LIN {X 0,Y 149.107,Z 804.963,A -85,B 0,C 180,E1 -24968.646,E2 -24968.646} C_VEL
LIN {X 0,Y 155.248,Z 796.631,A -85,B 0,C 180,E1 -24971.89,E2 -24971.89} C_VEL
LIN {X 0,Y 160.793,Z 788.072,A -85,B 0,C 180,E1 -24974.372,E2 -24974.372} C_VEL
LIN {X 0,Y 166.724,Z 777.561,A -85,B 0,C 180,E1 -24976.646,E2 -24976.646} C_VEL
LIN {X 0,Y 171.709,Z 767.159,A -85,B 0,C 180,E1 -24978.327,E2 -24978.327} C_VEL
LIN {X 0,Y 176.218,Z 755.637,A -85,B 0,C 180,E1 -24979.706,E2 -24979.706} C_VEL
LIN {X 0,Y 180.103,Z 742.538,A -85,B 0,C 180,E1 -24980.855,E2 -24980.855} C_VEL
LIN {X 0,Y 182.778,Z 729.709,A -85,B 0,C 180,E1 -24981.625,E2 -24981.625} C_VEL
LIN {X 0,Y 184.427,Z 715.563,A -85,B 0,C 180,E1 -24982.173,E2 -24982.173} C_VEL
LIN {X 0,Y 185.741,Z 699.59,A -85,B 0,C 180,E1 -24982.676,E2 -24982.676} C_VEL
LIN {X 0,Y 185.63,Z 687.899,A -85,B 0,C 180,E1 -24983.577,E2 -24983.577} C_VEL
LIN {X 0,Y 184.651,Z 684.228,A -85,B 0,C 180,E1 -24984.352,E2 -24984.352} C_VEL
LIN {X 0,Y 180.191,Z 675.322,A -85,B 0,C 180,E1 -24987.593,E2 -24987.593} C_VEL
LIN {X 0,Y 176.995,Z 669.722,A -85,B 0,C 180,E1 -24990.207,E2 -24990.207} C_VEL
LIN {X 0,Y 173.204,Z 663.907,A -85,B 0,C 180,E1 -24993.751,E2 -24993.751} C_VEL
LIN {X 0,Y 170.669,Z 660.092,A -85,B 0,C 180,E1 -24996.576,E2 -24996.576} C_VEL
LIN {X 0,Y 168.154,Z 656.304,A -85,B 0,C 180,E1 -24999.989,E2 -24999.989} C_VEL
LIN {X 0,Y 165.387,Z 652.572,A -85,B 0,C 180,E1 -25005.228,E2 -25005.228} C_VEL
LIN {X 0,Y 164.803,Z 650.964,A -85,B 0,C 180,E1 -25007.063,E2 -25007.063} C_VEL
LIN {X 0,Y 163.574,Z 650.195,A -85,B 0,C 180,E1 -25012.594,E2 -25012.594} C_VEL
LIN {X 0,Y 163.96,Z 650.175,A -85,B 0,C 180,E1 -25018.772,E2 -25018.772} C_VEL
LIN {X 0,Y 165.067,Z 651.088,A -85,B 0,C 180,E1 -25022.589,E2 -25022.589} C_VEL
LIN {X 0,Y 166.617,Z 654.282,A -85,B 0,C 180,E1 -25026.357,E2 -25026.357} C_VEL
LIN {X 0,Y 168.172,Z 656.106,A -85,B 0,C 180,E1 -25028.941,E2 -25028.941} C_VEL
LIN {X 0,Y 170.766,Z 660.079,A -85,B 0,C 180,E1 -25032.478,E2 -25032.478} C_VEL
LIN {X 0,Y 174.551,Z 665.825,A -85,B 0,C 180,E1 -25036.521,E2 -25036.521} C_VEL
LIN {X 0,Y 178.449,Z 672.031,A -85,B 0,C 180,E1 -25039.947,E2 -25039.947} C_VEL
LIN {X 0,Y 183.117,Z 680.317,A -85,B 0,C 180,E1 -25043.47,E2 -25043.47} C_VEL
LIN {X 0,Y 186.858,Z 687.514,A -85,B 0,C 180,E1 -25045.951,E2 -25045.951} C_VEL
LIN {X 0,Y 185.177,Z 708.656,A -85,B 0,C 180,E1 -25046.819,E2 -25046.819} C_VEL
LIN {X 0,Y 183.07,Z 721.345,A -85,B 0,C 180,E1 -25047.63,E2 -25047.63} C_VEL
LIN {X 0,Y 179.924,Z 734.079,A -85,B 0,C 180,E1 -25048.788,E2 -25048.788} C_VEL
LIN {X 0,Y 176.07,Z 745.896,A -85,B 0,C 180,E1 -25050.327,E2 -25050.327} C_VEL
LIN {X 0,Y 171.395,Z 757.092,A -85,B 0,C 180,E1 -25052.213,E2 -25052.213} C_VEL
LIN {X 0,Y 166.178,Z 767.268,A -85,B 0,C 180,E1 -25054.444,E2 -25054.444} C_VEL
LIN {X 0,Y 160.701,Z 776.286,A -85,B 0,C 180,E1 -25057.05,E2 -25057.05} C_VEL
LIN {X 0,Y 155.565,Z 783.661,A -85,B 0,C 180,E1 -25059.826,E2 -25059.826} C_VEL
LIN {X 0,Y 149.854,Z 790.842,A -85,B 0,C 180,E1 -25063.372,E2 -25063.372} C_VEL
LIN {X 0,Y 144.674,Z 796.477,A -85,B 0,C 180,E1 -25067.15,E2 -25067.15} C_VEL
LIN {X 0,Y 140.117,Z 800.824,A -85,B 0,C 180,E1 -25071.174,E2 -25071.174} C_VEL
LIN {X 0,Y 135.784,Z 804.333,A -85,B 0,C 180,E1 -25075.908,E2 -25075.908} C_VEL
LIN {X 0,Y 132.074,Z 806.745,A -85,B 0,C 180,E1 -25081.386,E2 -25081.386} C_VEL
LIN {X 0,Y 129.344,Z 807.693,A -85,B 0,C 180,E1 -25087.475,E2 -25087.475} C_VEL
LIN {X 0,Y 128.338,Z 807.582,A -85,B 0,C 180,E1 -25090.819,E2 -25090.819} C_VEL
LIN {X 0,Y 127.671,Z 807.045,A -85,B 0,C 180,E1 -25094.024,E2 -25094.024} C_VEL
LIN {X 0,Y 127.38,Z 806.076,A -85,B 0,C 180,E1 -25097.251,E2 -25097.251} C_VEL
LIN {X 0,Y 127.514,Z 803.466,A -85,B 0,C 180,E1 -25102.784,E2 -25102.784} C_VEL
LIN {X 0,Y 128.551,Z 799.409,A -85,B 0,C 180,E1 -25108.434,E2 -25108.434} C_VEL
LIN {X 0,Y 129.967,Z 794.796,A -85,B 0,C 180,E1 -25113.1,E2 -25113.1} C_VEL
LIN {X 0,Y 132.074,Z 788.942,A -85,B 0,C 180,E1 -25117.645,E2 -25117.645} C_VEL
LIN {X 0,Y 134.811,Z 781.651,A -85,B 0,C 180,E1 -25122.036,E2 -25122.036} C_VEL
LIN {X 0,Y 137.595,Z 774.209,A -85,B 0,C 180,E1 -25125.554,E2 -25125.554} C_VEL
LIN {X 0,Y 139.505,Z 769.017,A -85,B 0,C 180,E1 -25127.593,E2 -25127.593} C_VEL
LIN {X 0,Y 137.283,Z 767.608,A -85,B 0,C 180,E1 -25128.723,E2 -25128.723} C_VEL
LIN {X 0,Y 136.619,Z 766.743,A -85,B 0,C 180,E1 -25129.295,E2 -25129.295} C_VEL
LIN {X 0,Y 133.731,Z 776.449,A -85,B 0,C 180,E1 -25133.212,E2 -25133.212} C_VEL
LIN {X 0,Y 131.498,Z 784.057,A -85,B 0,C 180,E1 -25137.111,E2 -25137.111} C_VEL
LIN {X 0,Y 129.644,Z 790.883,A -85,B 0,C 180,E1 -25141.489,E2 -25141.489} C_VEL
LIN {X 0,Y 128.29,Z 796.393,A -85,B 0,C 180,E1 -25145.922,E2 -25145.922} C_VEL
LIN {X 0,Y 127.318,Z 801.706,A -85,B 0,C 180,E1 -25151.482,E2 -25151.482} C_VEL
LIN {X 0,Y 127.189,Z 804.837,A -85,B 0,C 180,E1 -25155.915,E2 -25155.915} C_VEL
LIN {X 0,Y 127.664,Z 807.177,A -85,B 0,C 180,E1 -25160.416,E2 -25160.416} C_VEL
LIN {X 0,Y 128.778,Z 808.735,A -85,B 0,C 180,E1 -25164.945,E2 -25164.945} C_VEL
LIN {X 0,Y 130.611,Z 809.478,A -85,B 0,C 180,E1 -25169.419,E2 -25169.419} C_VEL
LIN {X 0,Y 134.05,Z 809.144,A -85,B 0,C 180,E1 -25175.202,E2 -25175.202} C_VEL
LIN {X 0,Y 137.079,Z 808.116,A -85,B 0,C 180,E1 -25178.968,E2 -25178.968} C_VEL
LIN {X 0,Y 142.535,Z 805.212,A -85,B 0,C 180,E1 -25184.265,E2 -25184.265} C_VEL
LIN {X 0,Y 149.024,Z 800.693,A -85,B 0,C 180,E1 -25189.127,E2 -25189.127} C_VEL
LIN {X 0,Y 155.716,Z 794.938,A -85,B 0,C 180,E1 -25193.172,E2 -25193.172} C_VEL
LIN {X 0,Y 161.965,Z 788.671,A -85,B 0,C 180,E1 -25196.368,E2 -25196.368} C_VEL
LIN {X 0,Y 168.681,Z 780.891,A -85,B 0,C 180,E1 -25199.283,E2 -25199.283} C_VEL
LIN {X 0,Y 174.996,Z 772.214,A -85,B 0,C 180,E1 -25201.727,E2 -25201.727} C_VEL
LIN {X 0,Y 181.207,Z 762.147,A -85,B 0,C 180,E1 -25203.892,E2 -25203.892} C_VEL
LIN {X 0,Y 186.728,Z 751.431,A -85,B 0,C 180,E1 -25205.67,E2 -25205.67} C_VEL
LIN {X 0,Y 191.579,Z 739.672,A -85,B 0,C 180,E1 -25207.133,E2 -25207.133} C_VEL
LIN {X 0,Y 195.37,Z 727.803,A -85,B 0,C 180,E1 -25208.273,E2 -25208.273} C_VEL
LIN {X 0,Y 198.233,Z 715.512,A -85,B 0,C 180,E1 -25209.15,E2 -25209.15} C_VEL
LIN {X 0,Y 200.271,Z 701.906,A -85,B 0,C 180,E1 -25209.794,E2 -25209.794} C_VEL
LIN {X 0,Y 201.094,Z 695.258,A -85,B 0,C 180,E1 -25210.064,E2 -25210.064} C_VEL
LIN {X 0,Y 199.845,Z 692.673,A -85,B 0,C 180,E1 -25211.821,E2 -25211.821} C_VEL
LIN {X 0,Y 198.373,Z 689.434,A -85,B 0,C 180,E1 -25214.359,E2 -25214.359} C_VEL
LIN {X 0,Y 197.219,Z 686.711,A -85,B 0,C 180,E1 -25217.375,E2 -25217.375} C_VEL
LIN {X 0,Y 196.404,Z 686.119,A -85,B 0,C 180,E1 -25220.967,E2 -25220.967} C_VEL
LIN {X 0,Y 196.29,Z 687.002,A -85,B 0,C 180,E1 -25223.762,E2 -25223.762} C_VEL
LIN {X 0,Y 196.81,Z 690.184,A -85,B 0,C 180,E1 -25227.513,E2 -25227.513} C_VEL
LIN {X 0,Y 197.265,Z 692.099,A -85,B 0,C 180,E1 -25229.076,E2 -25229.076} C_VEL
LIN {X 0,Y 198.259,Z 696.239,A -85,B 0,C 180,E1 -25231.548,E2 -25231.548} C_VEL
LIN {X 0,Y 199.313,Z 700.889,A -85,B 0,C 180,E1 -25233.671,E2 -25233.671} C_VEL
LIN {X 0,Y 200.13,Z 704.559,A -85,B 0,C 180,E1 -25235.026,E2 -25235.026} C_VEL
LIN {X 0,Y 199.762,Z 708.061,A -85,B 0,C 180,E1 -25235.223,E2 -25235.223} C_VEL
LIN {X 0,Y 197.093,Z 725.443,A -85,B 0,C 180,E1 -25235.867,E2 -25235.867} C_VEL
LIN {X 0,Y 193.859,Z 738.295,A -85,B 0,C 180,E1 -25236.541,E2 -25236.541} C_VEL
LIN {X 0,Y 189.397,Z 751.371,A -85,B 0,C 180,E1 -25237.52,E2 -25237.52} C_VEL
LIN {X 0,Y 184.463,Z 762.701,A -85,B 0,C 180,E1 -25238.646,E2 -25238.646} C_VEL
LIN {X 0,Y 178.307,Z 774.287,A -85,B 0,C 180,E1 -25240.213,E2 -25240.213} C_VEL
LIN {X 0,Y 172.401,Z 783.818,A -85,B 0,C 180,E1 -25241.931,E2 -25241.931} C_VEL
LIN {X 0,Y 164.854,Z 794.256,A -85,B 0,C 180,E1 -25244.434,E2 -25244.434} C_VEL
LIN {X 0,Y 157.908,Z 802.647,A -85,B 0,C 180,E1 -25247.257,E2 -25247.257} C_VEL
LIN {X 0,Y 150.413,Z 810.603,A -85,B 0,C 180,E1 -25250.893,E2 -25250.893} C_VEL
LIN {X 0,Y 144.716,Z 816.086,A -85,B 0,C 180,E1 -25254.355,E2 -25254.355} C_VEL
LIN {X 0,Y 140.343,Z 819.929,A -85,B 0,C 180,E1 -25257.577,E2 -25257.577} C_VEL
LIN {X 0,Y 137.381,Z 821.943,A -85,B 0,C 180,E1 -25259.529,E2 -25259.529} C_VEL
LIN {X 0,Y 131.252,Z 824.616,A -85,B 0,C 180,E1 -25262.665,E2 -25262.665} C_VEL
LIN {X 0,Y 125.55,Z 826.525,A -85,B 0,C 180,E1 -25266.18,E2 -25266.18} C_VEL
LIN {X 0,Y 123.348,Z 827.286,A -85,B 0,C 180,E1 -25268.67,E2 -25268.67} C_VEL
LIN {X 0,Y 121.392,Z 828.217,A -85,B 0,C 180,E1 -25273.174,E2 -25273.174} C_VEL
LIN {X 0,Y 120.096,Z 828.286,A -85,B 0,C 180,E1 -25279.889,E2 -25279.889} C_VEL
LIN {X 0,Y 120.164,Z 827.608,A -85,B 0,C 180,E1 -25283.866,E2 -25283.866} C_VEL
LIN {X 0,Y 120.672,Z 826.255,A -85,B 0,C 180,E1 -25288.749,E2 -25288.749} C_VEL
LIN {X 0,Y 120.78,Z 826.749,A -85,B 0,C 180,E1 -25290,E2 -25290} C_VEL
LIN {X 0,Y 119.997,Z 828.128,A -85,B 0,C 180,E1 -25296.727,E2 -25296.727} C_VEL
LIN {X 0,Y 120.025,Z 828.23,A -85,B 0,C 180,E1 -25300.117,E2 -25300.117} C_VEL
LIN {X 0,Y 121.377,Z 827.211,A -85,B 0,C 180,E1 -25306.828,E2 -25306.828} C_VEL
LIN {X 0,Y 124.481,Z 824.663,A -85,B 0,C 180,E1 -25313.278,E2 -25313.278} C_VEL
LIN {X 0,Y 127.795,Z 821.642,A -85,B 0,C 180,E1 -25317.868,E2 -25317.868} C_VEL
LIN {X 0,Y 131.898,Z 817.615,A -85,B 0,C 180,E1 -25322.196,E2 -25322.196} C_VEL
LIN {X 0,Y 137.817,Z 811.485,A -85,B 0,C 180,E1 -25326.811,E2 -25326.811} C_VEL
LIN {X 0,Y 143.637,Z 804.821,A -85,B 0,C 180,E1 -25330.413,E2 -25330.413} C_VEL
LIN {X 0,Y 150.046,Z 796.598,A -85,B 0,C 180,E1 -25333.698,E2 -25333.698} C_VEL
LIN {X 0,Y 155.805,Z 788.196,A -85,B 0,C 180,E1 -25336.195,E2 -25336.195} C_VEL
LIN {X 0,Y 161.952,Z 777.839,A -85,B 0,C 180,E1 -25338.465,E2 -25338.465} C_VEL
LIN {X 0,Y 167.736,Z 766.224,A -85,B 0,C 180,E1 -25340.343,E2 -25340.343} C_VEL
LIN {X 0,Y 172.414,Z 754.582,A -85,B 0,C 180,E1 -25341.689,E2 -25341.689} C_VEL
LIN {X 0,Y 176.413,Z 741.361,A -85,B 0,C 180,E1 -25342.82,E2 -25342.82} C_VEL
LIN {X 0,Y 179.066,Z 728.861,A -85,B 0,C 180,E1 -25343.542,E2 -25343.542} C_VEL
LIN {X 0,Y 180.73,Z 714.959,A -85,B 0,C 180,E1 -25344.077,E2 -25344.077} C_VEL
LIN {X 0,Y 181.987,Z 699.437,A -85,B 0,C 180,E1 -25344.6,E2 -25344.6} C_VEL
LIN {X 0,Y 181.961,Z 690.827,A -85,B 0,C 180,E1 -25345.285,E2 -25345.285} C_VEL
LIN {X 0,Y 181.33,Z 688.674,A -85,B 0,C 180,E1 -25345.806,E2 -25345.806} C_VEL
LIN {X 0,Y 176.769,Z 679.156,A -85,B 0,C 180,E1 -25349.468,E2 -25349.468} C_VEL
LIN {X 0,Y 173.564,Z 673.777,A -85,B 0,C 180,E1 -25352.365,E2 -25352.365} C_VEL
LIN {X 0,Y 171.058,Z 669.808,A -85,B 0,C 180,E1 -25354.964,E2 -25354.964} C_VEL
LIN {X 0,Y 169.045,Z 666.616,A -85,B 0,C 180,E1 -25357.383,E2 -25357.383} C_VEL
LIN {X 0,Y 166.494,Z 662.608,A -85,B 0,C 180,E1 -25361.159,E2 -25361.159} C_VEL
LIN {X 0,Y 164.281,Z 659.446,A -85,B 0,C 180,E1 -25365.754,E2 -25365.754} C_VEL
LIN {X 0,Y 163.731,Z 657.95,A -85,B 0,C 180,E1 -25367.607,E2 -25367.607} C_VEL
LIN {X 0,Y 162.621,Z 657.234,A -85,B 0,C 180,E1 -25373.703,E2 -25373.703} C_VEL
LIN {X 0,Y 163.082,Z 657.223,A -85,B 0,C 180,E1 -25378.765,E2 -25378.765} C_VEL
LIN {X 0,Y 164.014,Z 658.078,A -85,B 0,C 180,E1 -25382.149,E2 -25382.149} C_VEL
LIN {X 0,Y 165.723,Z 661.5,A -85,B 0,C 180,E1 -25386.391,E2 -25386.391} C_VEL
LIN {X 0,Y 166.843,Z 662.912,A -85,B 0,C 180,E1 -25388.326,E2 -25388.326} C_VEL
LIN {X 0,Y 169.836,Z 667.73,A -85,B 0,C 180,E1 -25392.548,E2 -25392.548} C_VEL
LIN {X 0,Y 172.908,Z 672.59,A -85,B 0,C 180,E1 -25395.924,E2 -25395.924} C_VEL
LIN {X 0,Y 176.43,Z 678.545,A -85,B 0,C 180,E1 -25399.186,E2 -25399.186} C_VEL
LIN {X 0,Y 180.876,Z 686.728,A -85,B 0,C 180,E1 -25402.714,E2 -25402.714} C_VEL
LIN {X 0,Y 182.968,Z 691.206,A -85,B 0,C 180,E1 -25404.238,E2 -25404.238} C_VEL
LIN {X 0,Y 181.385,Z 709.15,A -85,B 0,C 180,E1 -25404.956,E2 -25404.956} C_VEL
LIN {X 0,Y 179.198,Z 721.822,A -85,B 0,C 180,E1 -25405.751,E2 -25405.751} C_VEL
LIN {X 0,Y 175.873,Z 734.809,A -85,B 0,C 180,E1 -25406.925,E2 -25406.925} C_VEL
LIN {X 0,Y 171.872,Z 746.601,A -85,B 0,C 180,E1 -25408.462,E2 -25408.462} C_VEL
LIN {X 0,Y 167.031,Z 757.719,A -85,B 0,C 180,E1 -25410.326,E2 -25410.326} C_VEL
LIN {X 0,Y 162.168,Z 766.937,A -85,B 0,C 180,E1 -25412.321,E2 -25412.321} C_VEL
LIN {X 0,Y 156.404,Z 776.136,A -85,B 0,C 180,E1 -25414.911,E2 -25414.911} C_VEL
LIN {X 0,Y 149.945,Z 784.988,A -85,B 0,C 180,E1 -25418.274,E2 -25418.274} C_VEL
LIN {X 0,Y 143.982,Z 792,A -85,B 0,C 180,E1 -25421.896,E2 -25421.896} C_VEL
LIN {X 0,Y 137.699,Z 798.306,A -85,B 0,C 180,E1 -25426.449,E2 -25426.449} C_VEL
LIN {X 0,Y 133.013,Z 802.363,A -85,B 0,C 180,E1 -25430.652,E2 -25430.652} C_VEL
LIN {X 0,Y 129.446,Z 804.984,A -85,B 0,C 180,E1 -25434.528,E2 -25434.528} C_VEL
LIN {X 0,Y 125.713,Z 807.233,A -85,B 0,C 180,E1 -25439.792,E2 -25439.792} C_VEL
LIN {X 0,Y 123.962,Z 807.988,A -85,B 0,C 180,E1 -25443.028,E2 -25443.028} C_VEL
LIN {X 0,Y 122.497,Z 808.303,A -85,B 0,C 180,E1 -25446.631,E2 -25446.631} C_VEL
LIN {X 0,Y 120.727,Z 807.747,A -85,B 0,C 180,E1 -25453.078,E2 -25453.078} C_VEL
LIN {X 0,Y 120.342,Z 806.823,A -85,B 0,C 180,E1 -25456.491,E2 -25456.491} C_VEL
LIN {X 0,Y 120.425,Z 804.046,A -85,B 0,C 180,E1 -25462.804,E2 -25462.804} C_VEL
LIN {X 0,Y 121.402,Z 800.33,A -85,B 0,C 180,E1 -25468.341,E2 -25468.341} C_VEL
LIN {X 0,Y 122.869,Z 795.814,A -85,B 0,C 180,E1 -25473.279,E2 -25473.279} C_VEL
LIN {X 0,Y 125.441,Z 788.963,A -85,B 0,C 180,E1 -25478.863,E2 -25478.863} C_VEL
LIN {X 0,Y 128.429,Z 781.544,A -85,B 0,C 180,E1 -25483.448,E2 -25483.448} C_VEL
LIN {X 0,Y 131.428,Z 773.954,A -85,B 0,C 180,E1 -25487.104,E2 -25487.104} C_VEL
LIN {X 0,Y 132.095,Z 772.216,A -85,B 0,C 180,E1 -25487.813,E2 -25487.813} C_VEL
LIN {X 0,Y 129.648,Z 771.123,A -85,B 0,C 180,E1 -25488.98,E2 -25488.98} C_VEL
LIN {X 0,Y 128.834,Z 770.326,A -85,B 0,C 180,E1 -25489.697,E2 -25489.697} C_VEL
LIN {X 0,Y 126.012,Z 779.452,A -85,B 0,C 180,E1 -25493.85,E2 -25493.85} C_VEL
LIN {X 0,Y 123.52,Z 787.88,A -85,B 0,C 180,E1 -25498.804,E2 -25498.804} C_VEL
LIN {X 0,Y 121.586,Z 795.054,A -85,B 0,C 180,E1 -25504.302,E2 -25504.302} C_VEL
LIN {X 0,Y 120.4,Z 800.68,A -85,B 0,C 180,E1 -25509.947,E2 -25509.947} C_VEL
LIN {X 0,Y 120.092,Z 804.706,A -85,B 0,C 180,E1 -25515.391,E2 -25515.391} C_VEL
LIN {X 0,Y 120.512,Z 807.259,A -85,B 0,C 180,E1 -25520.096,E2 -25520.096} C_VEL
LIN {X 0,Y 121.543,Z 808.972,A -85,B 0,C 180,E1 -25524.674,E2 -25524.674} C_VEL
LIN {X 0,Y 123.246,Z 809.949,A -85,B 0,C 180,E1 -25529.121,E2 -25529.121} C_VEL
LIN {X 0,Y 125.601,Z 810.22,A -85,B 0,C 180,E1 -25533.541,E2 -25533.541} C_VEL
LIN {X 0,Y 128.819,Z 809.651,A -85,B 0,C 180,E1 -25538.04,E2 -25538.04} C_VEL
LIN {X 0,Y 132.75,Z 808.218,A -85,B 0,C 180,E1 -25542.35,E2 -25542.35} C_VEL
LIN {X 0,Y 137.371,Z 805.871,A -85,B 0,C 180,E1 -25546.417,E2 -25546.417} C_VEL
LIN {X 0,Y 142.63,Z 802.566,A -85,B 0,C 180,E1 -25550.219,E2 -25550.219} C_VEL
LIN {X 0,Y 148.462,Z 798.193,A -85,B 0,C 180,E1 -25553.767,E2 -25553.767} C_VEL
LIN {X 0,Y 155.617,Z 791.872,A -85,B 0,C 180,E1 -25557.412,E2 -25557.412} C_VEL
LIN {X 0,Y 161.64,Z 785.635,A -85,B 0,C 180,E1 -25560.044,E2 -25560.044} C_VEL
LIN {X 0,Y 168.871,Z 776.969,A -85,B 0,C 180,E1 -25562.809,E2 -25562.809} C_VEL
LIN {X 0,Y 175.8,Z 767.036,A -85,B 0,C 180,E1 -25565.172,E2 -25565.172} C_VEL
LIN {X 0,Y 181.924,Z 756.454,A -85,B 0,C 180,E1 -25567.07,E2 -25567.07} C_VEL
LIN {X 0,Y 187.312,Z 744.912,A -85,B 0,C 180,E1 -25568.632,E2 -25568.632} C_VEL
LIN {X 0,Y 191.713,Z 733.081,A -85,B 0,C 180,E1 -25569.855,E2 -25569.855} C_VEL
LIN {X 0,Y 195.284,Z 719.969,A -85,B 0,C 180,E1 -25570.882,E2 -25570.882} C_VEL
LIN {X 0,Y 197.665,Z 706.972,A -85,B 0,C 180,E1 -25571.574,E2 -25571.574} C_VEL
LIN {X 0,Y 198.609,Z 699.988,A -85,B 0,C 180,E1 -25571.843,E2 -25571.843} C_VEL
LIN {X 0,Y 196.923,Z 696.094,A -85,B 0,C 180,E1 -25574.946,E2 -25574.946} C_VEL
LIN {X 0,Y 195.909,Z 693.565,A -85,B 0,C 180,E1 -25577.831,E2 -25577.831} C_VEL
LIN {X 0,Y 195.249,Z 693.136,A -85,B 0,C 180,E1 -25581.097,E2 -25581.097} C_VEL
LIN {X 0,Y 195.144,Z 694.187,A -85,B 0,C 180,E1 -25583.911,E2 -25583.911} C_VEL
LIN {X 0,Y 195.747,Z 698.079,A -85,B 0,C 180,E1 -25588.008,E2 -25588.008} C_VEL
LIN {X 0,Y 196.607,Z 702.582,A -85,B 0,C 180,E1 -25590.758,E2 -25590.758} C_VEL
LIN {X 0,Y 197.649,Z 707.877,A -85,B 0,C 180,E1 -25593.122,E2 -25593.122} C_VEL
LIN {X 0,Y 197.642,Z 708.781,A -85,B 0,C 180,E1 -25593.282,E2 -25593.282} C_VEL
LIN {X 0,Y 194.999,Z 724.971,A -85,B 0,C 180,E1 -25593.875,E2 -25593.875} C_VEL
LIN {X 0,Y 191.326,Z 738.774,A -85,B 0,C 180,E1 -25594.576,E2 -25594.576} C_VEL
LIN {X 0,Y 186.726,Z 751.649,A -85,B 0,C 180,E1 -25595.521,E2 -25595.521} C_VEL
LIN {X 0,Y 180.917,Z 764.132,A -85,B 0,C 180,E1 -25596.756,E2 -25596.756} C_VEL
LIN {X 0,Y 174.586,Z 775.326,A -85,B 0,C 180,E1 -25598.284,E2 -25598.284} C_VEL
LIN {X 0,Y 167.816,Z 785.446,A -85,B 0,C 180,E1 -25600.158,E2 -25600.158} C_VEL
LIN {X 0,Y 160.012,Z 795.33,A -85,B 0,C 180,E1 -25602.636,E2 -25602.636} C_VEL
LIN {X 0,Y 152.81,Z 803.437,A -85,B 0,C 180,E1 -25605.464,E2 -25605.464} C_VEL
LIN {X 0,Y 145.004,Z 811.057,A -85,B 0,C 180,E1 -25609.134,E2 -25609.134} C_VEL
LIN {X 0,Y 138.998,Z 816.283,A -85,B 0,C 180,E1 -25612.647,E2 -25612.647} C_VEL
LIN {X 0,Y 133.716,Z 820.501,A -85,B 0,C 180,E1 -25616.505,E2 -25616.505} C_VEL
LIN {X 0,Y 129.257,Z 823.759,A -85,B 0,C 180,E1 -25620.703,E2 -25620.703} C_VEL
LIN {X 0,Y 124.501,Z 826.716,A -85,B 0,C 180,E1 -25626.726,E2 -25626.726} C_VEL
LIN {X 0,Y 123.348,Z 827.286,A -85,B 0,C 180,E1 -25628.67,E2 -25628.67} C_VEL
LIN {X 0,Y 121.415,Z 827.916,A -85,B 0,C 180,E1 -25631.271,E2 -25631.271} C_VEL
LIN {X 0,Y 117.164,Z 828.077,A -85,B 0,C 180,E1 -25635.574,E2 -25635.574} C_VEL
LIN {X 0,Y 114.221,Z 827.603,A -85,B 0,C 180,E1 -25639.222,E2 -25639.222} C_VEL
LIN {X 0,Y 113.127,Z 827.005,A -85,B 0,C 180,E1 -25642.137,E2 -25642.137} C_VEL
LIN {X 0,Y 113.093,Z 826.77,A -85,B 0,C 180,E1 -25643.13,E2 -25643.13} C_VEL
LIN {X 0,Y 113.568,Z 825.341,A -85,B 0,C 180,E1 -25648.227,E2 -25648.227} C_VEL
LIN {X 0,Y 113.693,Z 826.041,A -85,B 0,C 180,E1 -25650,E2 -25650} C_VEL
LIN {X 0,Y 113.005,Z 827.338,A -85,B 0,C 180,E1 -25655.691,E2 -25655.691} C_VEL
LIN {X 0,Y 113.004,Z 827.607,A -85,B 0,C 180,E1 -25660.753,E2 -25660.753} C_VEL
LIN {X 0,Y 113.567,Z 827.353,A -85,B 0,C 180,E1 -25664.331,E2 -25664.331} C_VEL
LIN {X 0,Y 116.044,Z 825.625,A -85,B 0,C 180,E1 -25671.307,E2 -25671.307} C_VEL
LIN {X 0,Y 117.946,Z 824.191,A -85,B 0,C 180,E1 -25674.651,E2 -25674.651} C_VEL
LIN {X 0,Y 121.956,Z 820.855,A -85,B 0,C 180,E1 -25679.971,E2 -25679.971} C_VEL
LIN {X 0,Y 127.586,Z 815.71,A -85,B 0,C 180,E1 -25685.336,E2 -25685.336} C_VEL
LIN {X 0,Y 134.148,Z 809.226,A -85,B 0,C 180,E1 -25689.923,E2 -25689.923} C_VEL
LIN {X 0,Y 140.459,Z 802.178,A -85,B 0,C 180,E1 -25693.47,E2 -25693.47} C_VEL
LIN {X 0,Y 147.354,Z 793.415,A -85,B 0,C 180,E1 -25696.663,E2 -25696.663} C_VEL
LIN {X 0,Y 153.516,Z 784.464,A -85,B 0,C 180,E1 -25699.057,E2 -25699.057} C_VEL
LIN {X 0,Y 159.337,Z 774.627,A -85,B 0,C 180,E1 -25701.021,E2 -25701.021} C_VEL
LIN {X 0,Y 164.676,Z 763.734,A -85,B 0,C 180,E1 -25702.641,E2 -25702.641} C_VEL
LIN {X 0,Y 169.502,Z 751.598,A -85,B 0,C 180,E1 -25703.95,E2 -25703.95} C_VEL
LIN {X 0,Y 173.207,Z 739.089,A -85,B 0,C 180,E1 -25704.944,E2 -25704.944} C_VEL
LIN {X 0,Y 175.857,Z 726.094,A -85,B 0,C 180,E1 -25705.633,E2 -25705.633} C_VEL
LIN {X 0,Y 177.692,Z 709.198,A -85,B 0,C 180,E1 -25706.229,E2 -25706.229} C_VEL
LIN {X 0,Y 178.421,Z 700.413,A -85,B 0,C 180,E1 -25706.533,E2 -25706.533} C_VEL
LIN {X 0,Y 178.45,Z 693.795,A -85,B 0,C 180,E1 -25707.076,E2 -25707.076} C_VEL
LIN {X 0,Y 174.248,Z 684.617,A -85,B 0,C 180,E1 -25710.722,E2 -25710.722} C_VEL
LIN {X 0,Y 171.392,Z 679.673,A -85,B 0,C 180,E1 -25713.505,E2 -25713.505} C_VEL
LIN {X 0,Y 169.197,Z 676.036,A -85,B 0,C 180,E1 -25715.96,E2 -25715.96} C_VEL
LIN {X 0,Y 167.398,Z 673.053,A -85,B 0,C 180,E1 -25718.286,E2 -25718.286} C_VEL
LIN {X 0,Y 165.24,Z 669.431,A -85,B 0,C 180,E1 -25721.728,E2 -25721.728} C_VEL
LIN {X 0,Y 163.188,Z 666.298,A -85,B 0,C 180,E1 -25726.298,E2 -25726.298} C_VEL
LIN {X 0,Y 162.706,Z 664.92,A -85,B 0,C 180,E1 -25728.063,E2 -25728.063} C_VEL
LIN {X 0,Y 161.835,Z 664.274,A -85,B 0,C 180,E1 -25732.514,E2 -25732.514} C_VEL
LIN {X 0,Y 162.338,Z 664.372,A -85,B 0,C 180,E1 -25739.38,E2 -25739.38} C_VEL
LIN {X 0,Y 162.97,Z 665.055,A -85,B 0,C 180,E1 -25741.699,E2 -25741.699} C_VEL
LIN {X 0,Y 164.833,Z 668.694,A -85,B 0,C 180,E1 -25746.426,E2 -25746.426} C_VEL
LIN {X 0,Y 165.599,Z 669.83,A -85,B 0,C 180,E1 -25747.816,E2 -25747.816} C_VEL
LIN {X 0,Y 168.286,Z 674.394,A -85,B 0,C 180,E1 -25751.844,E2 -25751.844} C_VEL
LIN {X 0,Y 171.084,Z 679.033,A -85,B 0,C 180,E1 -25755.105,E2 -25755.105} C_VEL
LIN {X 0,Y 174.169,Z 684.452,A -85,B 0,C 180,E1 -25758.148,E2 -25758.148} C_VEL
LIN {X 0,Y 178.413,Z 692.712,A -85,B 0,C 180,E1 -25761.748,E2 -25761.748} C_VEL
LIN {X 0,Y 179.166,Z 694.275,A -85,B 0,C 180,E1 -25762.334,E2 -25762.334} C_VEL
LIN {X 0,Y 177.771,Z 709.868,A -85,B 0,C 180,E1 -25763.017,E2 -25763.017} C_VEL
LIN {X 0,Y 175.434,Z 722.816,A -85,B 0,C 180,E1 -25763.83,E2 -25763.83} C_VEL
LIN {X 0,Y 172.169,Z 735.094,A -85,B 0,C 180,E1 -25764.927,E2 -25764.927} C_VEL
LIN {X 0,Y 168.497,Z 745.749,A -85,B 0,C 180,E1 -25766.267,E2 -25766.267} C_VEL
LIN {X 0,Y 163.928,Z 756.166,A -85,B 0,C 180,E1 -25767.93,E2 -25767.93} C_VEL
LIN {X 0,Y 158.383,Z 766.55,A -85,B 0,C 180,E1 -25770.088,E2 -25770.088} C_VEL
LIN {X 0,Y 152.339,Z 775.985,A -85,B 0,C 180,E1 -25772.656,E2 -25772.656} C_VEL
LIN {X 0,Y 145.54,Z 784.967,A -85,B 0,C 180,E1 -25776.019,E2 -25776.019} C_VEL
LIN {X 0,Y 139.21,Z 792.131,A -85,B 0,C 180,E1 -25779.658,E2 -25779.658} C_VEL
LIN {X 0,Y 134.342,Z 796.905,A -85,B 0,C 180,E1 -25782.914,E2 -25782.914} C_VEL
LIN {X 0,Y 129.05,Z 801.463,A -85,B 0,C 180,E1 -25787.1,E2 -25787.1} C_VEL
LIN {X 0,Y 124.466,Z 804.848,A -85,B 0,C 180,E1 -25791.603,E2 -25791.603} C_VEL
LIN {X 0,Y 121.797,Z 806.495,A -85,B 0,C 180,E1 -25794.76,E2 -25794.76} C_VEL
LIN {X 0,Y 119.459,Z 807.721,A -85,B 0,C 180,E1 -25798.03,E2 -25798.03} C_VEL
LIN {X 0,Y 117.505,Z 808.538,A -85,B 0,C 180,E1 -25801.415,E2 -25801.415} C_VEL
LIN {X 0,Y 115.653,Z 808.916,A -85,B 0,C 180,E1 -25805.717,E2 -25805.717} C_VEL
LIN {X 0,Y 113.816,Z 808.423,A -85,B 0,C 180,E1 -25812.017,E2 -25812.017} C_VEL
LIN {X 0,Y 113.326,Z 807.567,A -85,B 0,C 180,E1 -25815.637,E2 -25815.637} C_VEL
LIN {X 0,Y 113.171,Z 806.28,A -85,B 0,C 180,E1 -25819.263,E2 -25819.263} C_VEL
LIN {X 0,Y 113.59,Z 803.574,A -85,B 0,C 180,E1 -25824.675,E2 -25824.675} C_VEL
LIN {X 0,Y 114.705,Z 799.857,A -85,B 0,C 180,E1 -25830,E2 -25830} C_VEL
LIN {X 0,Y 116.441,Z 795.04,A -85,B 0,C 180,E1 -25835.194,E2 -25835.194} C_VEL
LIN {X 0,Y 118.89,Z 788.973,A -85,B 0,C 180,E1 -25840.215,E2 -25840.215} C_VEL
LIN {X 0,Y 122.134,Z 781.396,A -85,B 0,C 180,E1 -25845.007,E2 -25845.007} C_VEL
LIN {X 0,Y 124.007,Z 776.898,A -85,B 0,C 180,E1 -25847.31,E2 -25847.31} C_VEL
LIN {X 0,Y 124.312,Z 775.369,A -85,B 0,C 180,E1 -25848.116,E2 -25848.116} C_VEL
LIN {X 0,Y 122.4,Z 774.746,A -85,B 0,C 180,E1 -25848.999,E2 -25848.999} C_VEL
LIN {X 0,Y 121.067,Z 773.5,A -85,B 0,C 180,E1 -25850.071,E2 -25850.071} C_VEL
LIN {X 0,Y 118.228,Z 782.26,A -85,B 0,C 180,E1 -25854.589,E2 -25854.589} C_VEL
LIN {X 0,Y 116.256,Z 788.945,A -85,B 0,C 180,E1 -25858.921,E2 -25858.921} C_VEL
LIN {X 0,Y 114.677,Z 794.639,A -85,B 0,C 180,E1 -25863.474,E2 -25863.474} C_VEL
LIN {X 0,Y 113.303,Z 800.953,A -85,B 0,C 180,E1 -25869.996,E2 -25869.996} C_VEL
LIN {X 0,Y 112.995,Z 804.592,A -85,B 0,C 180,E1 -25875.005,E2 -25875.005} C_VEL
LIN {X 0,Y 113.704,Z 808.174,A -85,B 0,C 180,E1 -25881.823,E2 -25881.823} C_VEL
LIN {X 0,Y 115.655,Z 810.189,A -85,B 0,C 180,E1 -25888.29,E2 -25888.29} C_VEL
LIN {X 0,Y 118.073,Z 810.872,A -85,B 0,C 180,E1 -25893.229,E2 -25893.229} C_VEL
LIN {X 0,Y 121.297,Z 810.72,A -85,B 0,C 180,E1 -25897.975,E2 -25897.975} C_VEL
LIN {X 0,Y 126.64,Z 809.199,A -85,B 0,C 180,E1 -25903.89,E2 -25903.89} C_VEL
LIN {X 0,Y 133.247,Z 806.149,A -85,B 0,C 180,E1 -25909.354,E2 -25909.354} C_VEL
LIN {X 0,Y 140.921,Z 801.366,A -85,B 0,C 180,E1 -25914.276,E2 -25914.276} C_VEL
LIN {X 0,Y 148.303,Z 795.731,A -85,B 0,C 180,E1 -25918.08,E2 -25918.08} C_VEL
LIN {X 0,Y 155.347,Z 789.359,A -85,B 0,C 180,E1 -25921.198,E2 -25921.198} C_VEL
LIN {X 0,Y 162.812,Z 781.394,A -85,B 0,C 180,E1 -25923.992,E2 -25923.992} C_VEL
LIN {X 0,Y 169.69,Z 772.67,A -85,B 0,C 180,E1 -25926.294,E2 -25926.294} C_VEL
LIN {X 0,Y 176.324,Z 762.723,A -85,B 0,C 180,E1 -25928.288,E2 -25928.288} C_VEL
LIN {X 0,Y 182.376,Z 751.648,A -85,B 0,C 180,E1 -25929.986,E2 -25929.986} C_VEL
LIN {X 0,Y 187.53,Z 739.905,A -85,B 0,C 180,E1 -25931.324,E2 -25931.324} C_VEL
LIN {X 0,Y 191.538,Z 728.069,A -85,B 0,C 180,E1 -25932.363,E2 -25932.363} C_VEL
LIN {X 0,Y 194.349,Z 716.662,A -85,B 0,C 180,E1 -25933.116,E2 -25933.116} C_VEL
LIN {X 0,Y 196.252,Z 704.967,A -85,B 0,C 180,E1 -25933.721,E2 -25933.721} C_VEL
LIN {X 0,Y 195.472,Z 702.744,A -85,B 0,C 180,E1 -25935.584,E2 -25935.584} C_VEL
LIN {X 0,Y 194.722,Z 700.562,A -85,B 0,C 180,E1 -25937.943,E2 -25937.943} C_VEL
LIN {X 0,Y 194.093,Z 700.164,A -85,B 0,C 180,E1 -25941.229,E2 -25941.229} C_VEL
LIN {X 0,Y 193.981,Z 701.483,A -85,B 0,C 180,E1 -25944.063,E2 -25944.063} C_VEL
LIN {X 0,Y 194.382,Z 704.807,A -85,B 0,C 180,E1 -25947.423,E2 -25947.423} C_VEL
LIN {X 0,Y 194.977,Z 708.854,A -85,B 0,C 180,E1 -25949.89,E2 -25949.89} C_VEL
LIN {X 0,Y 195.492,Z 712.009,A -85,B 0,C 180,E1 -25951.347,E2 -25951.347} C_VEL
LIN {X 0,Y 193.071,Z 725.426,A -85,B 0,C 180,E1 -25951.865,E2 -25951.865} C_VEL
LIN {X 0,Y 189.186,Z 739.217,A -85,B 0,C 180,E1 -25952.547,E2 -25952.547} C_VEL
LIN {X 0,Y 184.284,Z 752.06,A -85,B 0,C 180,E1 -25953.465,E2 -25953.465} C_VEL
LIN {X 0,Y 178.313,Z 764.233,A -85,B 0,C 180,E1 -25954.64,E2 -25954.64} C_VEL
LIN {X 0,Y 171.776,Z 775.259,A -85,B 0,C 180,E1 -25956.096,E2 -25956.096} C_VEL
LIN {X 0,Y 164.753,Z 785.247,A -85,B 0,C 180,E1 -25957.894,E2 -25957.894} C_VEL
LIN {X 0,Y 156.641,Z 795.037,A -85,B 0,C 180,E1 -25960.295,E2 -25960.295} C_VEL
LIN {X 0,Y 149.093,Z 803.016,A -85,B 0,C 180,E1 -25963.061,E2 -25963.061} C_VEL
LIN {X 0,Y 141.982,Z 809.585,A -85,B 0,C 180,E1 -25966.134,E2 -25966.134} C_VEL
LIN {X 0,Y 135.452,Z 814.96,A -85,B 0,C 180,E1 -25969.567,E2 -25969.567} C_VEL
LIN {X 0,Y 129.607,Z 819.262,A -85,B 0,C 180,E1 -25973.383,E2 -25973.383} C_VEL
LIN {X 0,Y 123.759,Z 823.154,A -85,B 0,C 180,E1 -25978.41,E2 -25978.41} C_VEL
LIN {X 0,Y 120.36,Z 825.103,A -85,B 0,C 180,E1 -25982.152,E2 -25982.152} C_VEL
LIN {X 0,Y 116.04,Z 827.136,A -85,B 0,C 180,E1 -25988.692,E2 -25988.692} C_VEL
LIN {X 0,Y 113.623,Z 827.718,A -85,B 0,C 180,E1 -25995.676,E2 -25995.676} C_VEL
LIN {X 0,Y 113.093,Z 826.77,A -85,B 0,C 180,E1 -26003.13,E2 -26003.13} C_VEL
LIN {X 0,Y 112.856,Z 826.435,A -85,B 0,C 180,E1 -26005.106,E2 -26005.106} C_VEL
LIN {X 0,Y 111.502,Z 826.238,A -85,B 0,C 180,E1 -26008.045,E2 -26008.045} C_VEL
LIN {X 0,Y 106.132,Z 826.814,A -85,B 0,C 180,E1 -26017.215,E2 -26017.215} C_VEL
LIN {X 0,Y 105.866,Z 826.898,A -85,B 0,C 180,E1 -26019.404,E2 -26019.404} C_VEL
LIN {X 0,Y 106.673,Z 826.772,A -85,B 0,C 180,E1 -26025.28,E2 -26025.28} C_VEL
LIN {X 0,Y 107.769,Z 826.142,A -85,B 0,C 180,E1 -26029.03,E2 -26029.03} C_VEL
LIN {X 0,Y 111.486,Z 823.717,A -85,B 0,C 180,E1 -26036.185,E2 -26036.185} C_VEL
LIN {X 0,Y 116.167,Z 820.182,A -85,B 0,C 180,E1 -26042.114,E2 -26042.114} C_VEL
LIN {X 0,Y 121.839,Z 815.406,A -85,B 0,C 180,E1 -26047.276,E2 -26047.276} C_VEL
LIN {X 0,Y 128.766,Z 808.998,A -85,B 0,C 180,E1 -26051.958,E2 -26051.958} C_VEL
LIN {X 0,Y 135.377,Z 802.068,A -85,B 0,C 180,E1 -26055.545,E2 -26055.545} C_VEL
LIN {X 0,Y 142.577,Z 793.431,A -85,B 0,C 180,E1 -26058.737,E2 -26058.737} C_VEL
LIN {X 0,Y 148.967,Z 784.61,A -85,B 0,C 180,E1 -26061.116,E2 -26061.116} C_VEL
LIN {X 0,Y 154.979,Z 774.946,A -85,B 0,C 180,E1 -26063.057,E2 -26063.057} C_VEL
LIN {X 0,Y 160.492,Z 764.357,A -85,B 0,C 180,E1 -26064.644,E2 -26064.644} C_VEL
LIN {X 0,Y 165.443,Z 752.539,A -85,B 0,C 180,E1 -26065.928,E2 -26065.928} C_VEL
LIN {X 0,Y 169.341,Z 740.318,A -85,B 0,C 180,E1 -26066.916,E2 -26066.916} C_VEL
LIN {X 0,Y 172.245,Z 727.426,A -85,B 0,C 180,E1 -26067.621,E2 -26067.621} C_VEL
LIN {X 0,Y 174.045,Z 713.18,A -85,B 0,C 180,E1 -26068.147,E2 -26068.147} C_VEL
LIN {X 0,Y 175.09,Z 701.271,A -85,B 0,C 180,E1 -26068.546,E2 -26068.546} C_VEL
LIN {X 0,Y 175.107,Z 697.562,A -85,B 0,C 180,E1 -26068.877,E2 -26068.877} C_VEL
LIN {X 0,Y 171.593,Z 689.679,A -85,B 0,C 180,E1 -26072.232,E2 -26072.232} C_VEL
LIN {X 0,Y 168.288,Z 683.6,A -85,B 0,C 180,E1 -26075.877,E2 -26075.877} C_VEL
LIN {X 0,Y 165.844,Z 679.567,A -85,B 0,C 180,E1 -26079.13,E2 -26079.13} C_VEL
LIN {X 0,Y 163.878,Z 676.144,A -85,B 0,C 180,E1 -26082.53,E2 -26082.53} C_VEL
LIN {X 0,Y 161.948,Z 672.613,A -85,B 0,C 180,E1 -26087.468,E2 -26087.468} C_VEL
LIN {X 0,Y 161.64,Z 671.857,A -85,B 0,C 180,E1 -26088.717,E2 -26088.717} C_VEL
LIN {X 0,Y 160.965,Z 671.328,A -85,B 0,C 180,E1 -26092.473,E2 -26092.473} C_VEL
LIN {X 0,Y 161.459,Z 671.425,A -85,B 0,C 180,E1 -26099.376,E2 -26099.376} C_VEL
LIN {X 0,Y 161.954,Z 672.043,A -85,B 0,C 180,E1 -26101.297,E2 -26101.297} C_VEL
LIN {X 0,Y 163.822,Z 675.753,A -85,B 0,C 180,E1 -26106.234,E2 -26106.234} C_VEL
LIN {X 0,Y 164.483,Z 677.003,A -85,B 0,C 180,E1 -26107.519,E2 -26107.519} C_VEL
LIN {X 0,Y 166.683,Z 680.89,A -85,B 0,C 180,E1 -26111.013,E2 -26111.013} C_VEL
LIN {X 0,Y 169.236,Z 685.338,A -85,B 0,C 180,E1 -26114.198,E2 -26114.198} C_VEL
LIN {X 0,Y 172.311,Z 691.122,A -85,B 0,C 180,E1 -26117.429,E2 -26117.429} C_VEL
LIN {X 0,Y 175.675,Z 698.027,A -85,B 0,C 180,E1 -26120.483,E2 -26120.483} C_VEL
LIN {X 0,Y 173.982,Z 713.054,A -85,B 0,C 180,E1 -26121.127,E2 -26121.127} C_VEL
LIN {X 0,Y 171.626,Z 724.974,A -85,B 0,C 180,E1 -26121.919,E2 -26121.919} C_VEL
LIN {X 0,Y 168.039,Z 737.354,A -85,B 0,C 180,E1 -26123.06,E2 -26123.06} C_VEL
LIN {X 0,Y 163.39,Z 749.649,A -85,B 0,C 180,E1 -26124.682,E2 -26124.682} C_VEL
LIN {X 0,Y 158.996,Z 758.851,A -85,B 0,C 180,E1 -26126.233,E2 -26126.233} C_VEL
LIN {X 0,Y 153.573,Z 768.32,A -85,B 0,C 180,E1 -26128.246,E2 -26128.246} C_VEL
LIN {X 0,Y 147.306,Z 777.479,A -85,B 0,C 180,E1 -26130.822,E2 -26130.822} C_VEL
LIN {X 0,Y 140.217,Z 786.306,A -85,B 0,C 180,E1 -26134.208,E2 -26134.208} C_VEL
LIN {X 0,Y 133.604,Z 793.291,A -85,B 0,C 180,E1 -26137.905,E2 -26137.905} C_VEL
LIN {X 0,Y 127.356,Z 798.919,A -85,B 0,C 180,E1 -26142.045,E2 -26142.045} C_VEL
LIN {X 0,Y 122.054,Z 803.019,A -85,B 0,C 180,E1 -26146.294,E2 -26146.294} C_VEL
LIN {X 0,Y 117.014,Z 806.296,A -85,B 0,C 180,E1 -26151.334,E2 -26151.334} C_VEL
LIN {X 0,Y 113.333,Z 808.208,A -85,B 0,C 180,E1 -26156.076,E2 -26156.076} C_VEL
LIN {X 0,Y 111.162,Z 809.064,A -85,B 0,C 180,E1 -26159.617,E2 -26159.617} C_VEL
LIN {X 0,Y 108.856,Z 809.527,A -85,B 0,C 180,E1 -26164.672,E2 -26164.672} C_VEL
LIN {X 0,Y 106.951,Z 809.094,A -85,B 0,C 180,E1 -26170.819,E2 -26170.819} C_VEL
LIN {X 0,Y 106.325,Z 808.304,A -85,B 0,C 180,E1 -26174.669,E2 -26174.669} C_VEL
LIN {X 0,Y 106.096,Z 807.061,A -85,B 0,C 180,E1 -26178.538,E2 -26178.538} C_VEL
LIN {X 0,Y 106.262,Z 805.226,A -85,B 0,C 180,E1 -26182.785,E2 -26182.785} C_VEL
LIN {X 0,Y 107.095,Z 802.117,A -85,B 0,C 180,E1 -26188.12,E2 -26188.12} C_VEL
LIN {X 0,Y 108.668,Z 797.767,A -85,B 0,C 180,E1 -26193.708,E2 -26193.708} C_VEL
LIN {X 0,Y 111.048,Z 792.227,A -85,B 0,C 180,E1 -26199.103,E2 -26199.103} C_VEL
LIN {X 0,Y 114.084,Z 785.311,A -85,B 0,C 180,E1 -26204.265,E2 -26204.265} C_VEL
LIN {X 0,Y 116.561,Z 779.749,A -85,B 0,C 180,E1 -26207.546,E2 -26207.546} C_VEL
LIN {X 0,Y 114.72,Z 777.907,A -85,B 0,C 180,E1 -26209.29,E2 -26209.29} C_VEL
LIN {X 0,Y 113.21,Z 776.696,A -85,B 0,C 180,E1 -26210.622,E2 -26210.622} C_VEL
LIN {X 0,Y 110.533,Z 784.932,A -85,B 0,C 180,E1 -26215.401,E2 -26215.401} C_VEL
LIN {X 0,Y 108.525,Z 791.39,A -85,B 0,C 180,E1 -26220.124,E2 -26220.124} C_VEL
LIN {X 0,Y 107.047,Z 796.935,A -85,B 0,C 180,E1 -26225.193,E2 -26225.193} C_VEL
LIN {X 0,Y 106.024,Z 802.322,A -85,B 0,C 180,E1 -26231.518,E2 -26231.518} C_VEL
LIN {X 0,Y 106.09,Z 806.678,A -85,B 0,C 180,E1 -26238.513,E2 -26238.513} C_VEL
LIN {X 0,Y 106.99,Z 809.039,A -85,B 0,C 180,E1 -26243.758,E2 -26243.758} C_VEL
LIN {X 0,Y 108.64,Z 810.624,A -85,B 0,C 180,E1 -26248.833,E2 -26248.833} C_VEL
LIN {X 0,Y 110.985,Z 811.432,A -85,B 0,C 180,E1 -26253.687,E2 -26253.687} C_VEL
LIN {X 0,Y 114.032,Z 811.562,A -85,B 0,C 180,E1 -26258.297,E2 -26258.297} C_VEL
LIN {X 0,Y 117.76,Z 811,A -85,B 0,C 180,E1 -26262.72,E2 -26262.72} C_VEL
LIN {X 0,Y 122.501,Z 809.536,A -85,B 0,C 180,E1 -26267.234,E2 -26267.234} C_VEL
LIN {X 0,Y 127.94,Z 807.175,A -85,B 0,C 180,E1 -26271.398,E2 -26271.398} C_VEL
LIN {X 0,Y 135.654,Z 802.889,A -85,B 0,C 180,E1 -26276.144,E2 -26276.144} C_VEL
LIN {X 0,Y 143.454,Z 797.453,A -85,B 0,C 180,E1 -26280,E2 -26280} C_VEL
LIN {X 0,Y 151.235,Z 790.91,A -85,B 0,C 180,E1 -26283.282,E2 -26283.282} C_VEL
LIN {X 0,Y 159.866,Z 782.266,A -85,B 0,C 180,E1 -26286.311,E2 -26286.311} C_VEL
LIN {X 0,Y 167.74,Z 772.741,A -85,B 0,C 180,E1 -26288.736,E2 -26288.736} C_VEL
LIN {X 0,Y 174.89,Z 762.264,A -85,B 0,C 180,E1 -26290.711,E2 -26290.711} C_VEL
LIN {X 0,Y 181.438,Z 750.341,A -85,B 0,C 180,E1 -26292.386,E2 -26292.386} C_VEL
LIN {X 0,Y 186.612,Z 738.468,A -85,B 0,C 180,E1 -26293.633,E2 -26293.633} C_VEL
LIN {X 0,Y 190.934,Z 725.264,A -85,B 0,C 180,E1 -26294.695,E2 -26294.695} C_VEL
LIN {X 0,Y 193.802,Z 712.805,A -85,B 0,C 180,E1 -26295.404,E2 -26295.404} C_VEL
LIN {X 0,Y 194.253,Z 709.957,A -85,B 0,C 180,E1 -26295.557,E2 -26295.557} C_VEL
LIN {X 0,Y 193.474,Z 707.47,A -85,B 0,C 180,E1 -26298.347,E2 -26298.347} C_VEL
LIN {X 0,Y 192.892,Z 707.266,A -85,B 0,C 180,E1 -26301.731,E2 -26301.731} C_VEL
LIN {X 0,Y 192.802,Z 708.673,A -85,B 0,C 180,E1 -26303.979,E2 -26303.979} C_VEL
LIN {X 0,Y 193.047,Z 711.59,A -85,B 0,C 180,E1 -26306.874,E2 -26306.874} C_VEL
LIN {X 0,Y 193.415,Z 715.282,A -85,B 0,C 180,E1 -26309.088,E2 -26309.088} C_VEL
LIN {X 0,Y 193.481,Z 716.011,A -85,B 0,C 180,E1 -26309.455,E2 -26309.455} C_VEL
LIN {X 0,Y 190.506,Z 729.408,A -85,B 0,C 180,E1 -26309.962,E2 -26309.962} C_VEL
LIN {X 0,Y 185.939,Z 743.371,A -85,B 0,C 180,E1 -26310.698,E2 -26310.698} C_VEL
LIN {X 0,Y 180.55,Z 755.894,A -85,B 0,C 180,E1 -26311.628,E2 -26311.628} C_VEL
LIN {X 0,Y 173.692,Z 768.391,A -85,B 0,C 180,E1 -26312.905,E2 -26312.905} C_VEL
LIN {X 0,Y 166.278,Z 779.51,A -85,B 0,C 180,E1 -26314.495,E2 -26314.495} C_VEL
LIN {X 0,Y 157.743,Z 790.164,A -85,B 0,C 180,E1 -26316.684,E2 -26316.684} C_VEL
LIN {X 0,Y 149.529,Z 798.929,A -85,B 0,C 180,E1 -26319.15,E2 -26319.15} C_VEL
LIN {X 0,Y 141.884,Z 806.07,A -85,B 0,C 180,E1 -26322.014,E2 -26322.014} C_VEL
LIN {X 0,Y 134.616,Z 811.93,A -85,B 0,C 180,E1 -26325.188,E2 -26325.188} C_VEL
LIN {X 0,Y 125.957,Z 818.028,A -85,B 0,C 180,E1 -26330.085,E2 -26330.085} C_VEL
LIN {X 0,Y 120.315,Z 821.503,A -85,B 0,C 180,E1 -26334.259,E2 -26334.259} C_VEL
LIN {X 0,Y 114.097,Z 824.786,A -85,B 0,C 180,E1 -26340.478,E2 -26340.478} C_VEL
LIN {X 0,Y 109.438,Z 826.587,A -85,B 0,C 180,E1 -26347.337,E2 -26347.337} C_VEL
LIN {X 0,Y 106.735,Z 826.949,A -85,B 0,C 180,E1 -26354.73,E2 -26354.73} C_VEL
LIN {X 0,Y 106.04,Z 825.913,A -85,B 0,C 180,E1 -26362.383,E2 -26362.383} C_VEL
LIN {X 0,Y 106.503,Z 824.428,A -85,B 0,C 180,E1 -26367.636,E2 -26367.636} C_VEL
LIN {X 0,Y 106.607,Z 825.316,A -85,B 0,C 180,E1 -26370,E2 -26370} C_VEL
LIN {X 0,Y 105.952,Z 826.615,A -85,B 0,C 180,E1 -26375.742,E2 -26375.742} C_VEL
LIN {X 0,Y 105.866,Z 826.898,A -85,B 0,C 180,E1 -26379.404,E2 -26379.404} C_VEL
LIN {X 0,Y 105.493,Z 826.924,A -85,B 0,C 180,E1 -26382.6,E2 -26382.6} C_VEL
LIN {X 0,Y 103.837,Z 826.177,A -85,B 0,C 180,E1 -26387.94,E2 -26387.94} C_VEL
LIN {X 0,Y 103.07,Z 825.18,A -85,B 0,C 180,E1 -26392.285,E2 -26392.285} C_VEL
LIN {X 0,Y 103.679,Z 824.192,A -85,B 0,C 180,E1 -26395.498,E2 -26395.498} C_VEL
LIN {X 0,Y 104.214,Z 823.764,A -85,B 0,C 180,E1 -26396.525,E2 -26396.525} C_VEL
LIN {X 0,Y 107.824,Z 821.481,A -85,B 0,C 180,E1 -26401.428,E2 -26401.428} C_VEL
LIN {X 0,Y 112.566,Z 817.997,A -85,B 0,C 180,E1 -26406.378,E2 -26406.378} C_VEL
LIN {X 0,Y 118.253,Z 813.471,A -85,B 0,C 180,E1 -26410.824,E2 -26410.824} C_VEL
LIN {X 0,Y 125.819,Z 806.665,A -85,B 0,C 180,E1 -26415.412,E2 -26415.412} C_VEL
LIN {X 0,Y 132.976,Z 799.306,A -85,B 0,C 180,E1 -26418.861,E2 -26418.861} C_VEL
LIN {X 0,Y 140.619,Z 790.209,A -85,B 0,C 180,E1 -26421.92,E2 -26421.92} C_VEL
LIN {X 0,Y 148.007,Z 779.721,A -85,B 0,C 180,E1 -26424.404,E2 -26424.404} C_VEL
LIN {X 0,Y 154.368,Z 769.076,A -85,B 0,C 180,E1 -26426.187,E2 -26426.187} C_VEL
LIN {X 0,Y 159.382,Z 758.742,A -85,B 0,C 180,E1 -26427.491,E2 -26427.491} C_VEL
LIN {X 0,Y 164.128,Z 746.398,A -85,B 0,C 180,E1 -26428.617,E2 -26428.617} C_VEL
LIN {X 0,Y 167.781,Z 733.457,A -85,B 0,C 180,E1 -26429.477,E2 -26429.477} C_VEL
LIN {X 0,Y 170.168,Z 720.434,A -85,B 0,C 180,E1 -26430.026,E2 -26430.026} C_VEL
LIN {X 0,Y 171.98,Z 702.164,A -85,B 0,C 180,E1 -26430.634,E2 -26430.634} C_VEL
LIN {X 0,Y 171.747,Z 701.077,A -85,B 0,C 180,E1 -26430.919,E2 -26430.919} C_VEL
LIN {X 0,Y 169.385,Z 695.409,A -85,B 0,C 180,E1 -26433.428,E2 -26433.428} C_VEL
LIN {X 0,Y 166.278,Z 689.547,A -85,B 0,C 180,E1 -26437.15,E2 -26437.15} C_VEL
LIN {X 0,Y 164.412,Z 686.171,A -85,B 0,C 180,E1 -26439.873,E2 -26439.873} C_VEL
LIN {X 0,Y 162.579,Z 682.839,A -85,B 0,C 180,E1 -26443.296,E2 -26443.296} C_VEL
LIN {X 0,Y 160.81,Z 679.09,A -85,B 0,C 180,E1 -26448.474,E2 -26448.474} C_VEL
LIN {X 0,Y 160.094,Z 678.382,A -85,B 0,C 180,E1 -26452.432,E2 -26452.432} C_VEL
LIN {X 0,Y 160.451,Z 678.349,A -85,B 0,C 180,E1 -26458.745,E2 -26458.745} C_VEL
LIN {X 0,Y 160.935,Z 679.013,A -85,B 0,C 180,E1 -26460.853,E2 -26460.853} C_VEL
LIN {X 0,Y 163.026,Z 683.305,A -85,B 0,C 180,E1 -26466.498,E2 -26466.498} C_VEL
LIN {X 0,Y 165.17,Z 687.44,A -85,B 0,C 180,E1 -26470.229,E2 -26470.229} C_VEL
LIN {X 0,Y 167.64,Z 692.042,A -85,B 0,C 180,E1 -26473.524,E2 -26473.524} C_VEL
LIN {X 0,Y 170.785,Z 698.326,A -85,B 0,C 180,E1 -26476.996,E2 -26476.996} C_VEL
LIN {X 0,Y 172.298,Z 701.661,A -85,B 0,C 180,E1 -26478.491,E2 -26478.491} C_VEL
LIN {X 0,Y 170.526,Z 715.484,A -85,B 0,C 180,E1 -26479.124,E2 -26479.124} C_VEL
LIN {X 0,Y 167.944,Z 727.226,A -85,B 0,C 180,E1 -26479.929,E2 -26479.929} C_VEL
LIN {X 0,Y 164.601,Z 738.134,A -85,B 0,C 180,E1 -26480.937,E2 -26480.937} C_VEL
LIN {X 0,Y 159.778,Z 750.399,A -85,B 0,C 180,E1 -26482.53,E2 -26482.53} C_VEL
LIN {X 0,Y 154.312,Z 761.243,A -85,B 0,C 180,E1 -26484.376,E2 -26484.376} C_VEL
LIN {X 0,Y 147.601,Z 771.955,A -85,B 0,C 180,E1 -26486.778,E2 -26486.778} C_VEL
LIN {X 0,Y 140.915,Z 780.898,A -85,B 0,C 180,E1 -26489.509,E2 -26489.509} C_VEL
LIN {X 0,Y 133.854,Z 788.858,A -85,B 0,C 180,E1 -26492.854,E2 -26492.854} C_VEL
LIN {X 0,Y 127.018,Z 795.446,A -85,B 0,C 180,E1 -26496.652,E2 -26496.652} C_VEL
LIN {X 0,Y 120.724,Z 800.624,A -85,B 0,C 180,E1 -26500.819,E2 -26500.819} C_VEL
LIN {X 0,Y 115.086,Z 804.559,A -85,B 0,C 180,E1 -26505.392,E2 -26505.392} C_VEL
LIN {X 0,Y 110.17,Z 807.394,A -85,B 0,C 180,E1 -26510.364,E2 -26510.364} C_VEL
LIN {X 0,Y 107.353,Z 808.697,A -85,B 0,C 180,E1 -26513.901,E2 -26513.901} C_VEL
LIN {X 0,Y 104.945,Z 809.589,A -85,B 0,C 180,E1 -26517.606,E2 -26517.606} C_VEL
LIN {X 0,Y 102.076,Z 810.14,A -85,B 0,C 180,E1 -26523.516,E2 -26523.516} C_VEL
LIN {X 0,Y 100.145,Z 809.764,A -85,B 0,C 180,E1 -26529.459,E2 -26529.459} C_VEL
LIN {X 0,Y 99.376,Z 809.015,A -85,B 0,C 180,E1 -26533.568,E2 -26533.568} C_VEL
LIN {X 0,Y 99.033,Z 807.842,A -85,B 0,C 180,E1 -26537.708,E2 -26537.708} C_VEL
LIN {X 0,Y 99.184,Z 805.824,A -85,B 0,C 180,E1 -26542.756,E2 -26542.756} C_VEL
LIN {X 0,Y 100.417,Z 801.723,A -85,B 0,C 180,E1 -26550,E2 -26550} C_VEL
LIN {X 0,Y 102.294,Z 797.071,A -85,B 0,C 180,E1 -26555.915,E2 -26555.915} C_VEL
LIN {X 0,Y 104.989,Z 791.185,A -85,B 0,C 180,E1 -26561.585,E2 -26561.585} C_VEL
LIN {X 0,Y 108.512,Z 783.852,A -85,B 0,C 180,E1 -26566.944,E2 -26566.944} C_VEL
LIN {X 0,Y 109.179,Z 782.478,A -85,B 0,C 180,E1 -26567.804,E2 -26567.804} C_VEL
LIN {X 0,Y 108.294,Z 781.312,A -85,B 0,C 180,E1 -26568.934,E2 -26568.934} C_VEL
LIN {X 0,Y 105.4,Z 779.687,A -85,B 0,C 180,E1 -26571.235,E2 -26571.235} C_VEL
LIN {X 0,Y 102.544,Z 788.275,A -85,B 0,C 180,E1 -26577.004,E2 -26577.004} C_VEL
LIN {X 0,Y 100.498,Z 795.127,A -85,B 0,C 180,E1 -26582.946,E2 -26582.946} C_VEL
LIN {X 0,Y 99.125,Z 801.041,A -85,B 0,C 180,E1 -26589.649,E2 -26589.649} C_VEL
LIN {X 0,Y 98.825,Z 804.937,A -85,B 0,C 180,E1 -26595.328,E2 -26595.328} C_VEL
LIN {X 0,Y 99.317,Z 807.996,A -85,B 0,C 180,E1 -26601.112,E2 -26601.112} C_VEL
LIN {X 0,Y 100.692,Z 810.213,A -85,B 0,C 180,E1 -26606.881,E2 -26606.881} C_VEL
LIN {X 0,Y 103.004,Z 811.632,A -85,B 0,C 180,E1 -26612.495,E2 -26612.495} C_VEL
LIN {X 0,Y 106.201,Z 812.265,A -85,B 0,C 180,E1 -26617.887,E2 -26617.887} C_VEL
LIN {X 0,Y 110.243,Z 812.092,A -85,B 0,C 180,E1 -26622.984,E2 -26622.984} C_VEL
LIN {X 0,Y 115.072,Z 811.057,A -85,B 0,C 180,E1 -26627.733,E2 -26627.733} C_VEL
LIN {X 0,Y 122.501,Z 808.383,A -85,B 0,C 180,E1 -26633.411,E2 -26633.411} C_VEL
LIN {X 0,Y 131.062,Z 804.068,A -85,B 0,C 180,E1 -26638.429,E2 -26638.429} C_VEL
LIN {X 0,Y 139.05,Z 798.967,A -85,B 0,C 180,E1 -26642.172,E2 -26642.172} C_VEL
LIN {X 0,Y 147.366,Z 792.517,A -85,B 0,C 180,E1 -26645.473,E2 -26645.473} C_VEL
LIN {X 0,Y 156.298,Z 784.207,A -85,B 0,C 180,E1 -26648.423,E2 -26648.423} C_VEL
LIN {X 0,Y 163.655,Z 775.962,A -85,B 0,C 180,E1 -26650.559,E2 -26650.559} C_VEL
LIN {X 0,Y 171.723,Z 765.033,A -85,B 0,C 180,E1 -26652.655,E2 -26652.655} C_VEL
LIN {X 0,Y 178.269,Z 754.216,A -85,B 0,C 180,E1 -26654.218,E2 -26654.218} C_VEL
LIN {X 0,Y 184.051,Z 742.157,A -85,B 0,C 180,E1 -26655.503,E2 -26655.503} C_VEL
LIN {X 0,Y 188.483,Z 730.195,A -85,B 0,C 180,E1 -26656.491,E2 -26656.491} C_VEL
LIN {X 0,Y 191.582,Z 718.838,A -85,B 0,C 180,E1 -26657.196,E2 -26657.196} C_VEL
LIN {X 0,Y 192.275,Z 715.486,A -85,B 0,C 180,E1 -26657.386,E2 -26657.386} C_VEL
LIN {X 0,Y 192.155,Z 714.458,A -85,B 0,C 180,E1 -26658.489,E2 -26658.489} C_VEL
LIN {X 0,Y 191.689,Z 714.211,A -85,B 0,C 180,E1 -26661.508,E2 -26661.508} C_VEL
LIN {X 0,Y 191.538,Z 715.423,A -85,B 0,C 180,E1 -26663.467,E2 -26663.467} C_VEL
LIN {X 0,Y 191.52,Z 718.044,A -85,B 0,C 180,E1 -26666.126,E2 -26666.126} C_VEL
LIN {X 0,Y 191.615,Z 720.063,A -85,B 0,C 180,E1 -26667.471,E2 -26667.471} C_VEL
LIN {X 0,Y 188.192,Z 733.161,A -85,B 0,C 180,E1 -26668.014,E2 -26668.014} C_VEL
LIN {X 0,Y 184.109,Z 744.498,A -85,B 0,C 180,E1 -26668.603,E2 -26668.603} C_VEL
LIN {X 0,Y 178.578,Z 756.461,A -85,B 0,C 180,E1 -26669.458,E2 -26669.458} C_VEL
LIN {X 0,Y 171.561,Z 768.646,A -85,B 0,C 180,E1 -26670.656,E2 -26670.656} C_VEL
LIN {X 0,Y 163.936,Z 779.537,A -85,B 0,C 180,E1 -26672.149,E2 -26672.149} C_VEL
LIN {X 0,Y 155.13,Z 790.085,A -85,B 0,C 180,E1 -26674.231,E2 -26674.231} C_VEL
LIN {X 0,Y 146.557,Z 798.69,A -85,B 0,C 180,E1 -26676.562,E2 -26676.562} C_VEL
LIN {X 0,Y 137.257,Z 806.71,A -85,B 0,C 180,E1 -26679.823,E2 -26679.823} C_VEL
LIN {X 0,Y 129.695,Z 812.318,A -85,B 0,C 180,E1 -26682.986,E2 -26682.986} C_VEL
LIN {X 0,Y 122.762,Z 816.842,A -85,B 0,C 180,E1 -26686.609,E2 -26686.609} C_VEL
LIN {X 0,Y 114.604,Z 821.401,A -85,B 0,C 180,E1 -26692.177,E2 -26692.177} C_VEL
LIN {X 0,Y 107.949,Z 824.432,A -85,B 0,C 180,E1 -26698.612,E2 -26698.612} C_VEL
LIN {X 0,Y 102.908,Z 825.998,A -85,B 0,C 180,E1 -26705.811,E2 -26705.811} C_VEL
LIN {X 0,Y 99.871,Z 826.183,A -85,B 0,C 180,E1 -26713.652,E2 -26713.652} C_VEL
LIN {X 0,Y 99.026,Z 824.917,A -85,B 0,C 180,E1 -26721.84,E2 -26721.84} C_VEL
LIN {X 0,Y 99.417,Z 823.467,A -85,B 0,C 180,E1 -26726.961,E2 -26726.961} C_VEL
LIN {X 0,Y 99.524,Z 824.578,A -85,B 0,C 180,E1 -26730,E2 -26730} C_VEL
LIN {X 0,Y 98.893,Z 825.872,A -85,B 0,C 180,E1 -26735.765,E2 -26735.765} C_VEL
LIN {X 0,Y 99.03,Z 826.361,A -85,B 0,C 180,E1 -26742.292,E2 -26742.292} C_VEL
LIN {X 0,Y 101.039,Z 825.606,A -85,B 0,C 180,E1 -26750.351,E2 -26750.351} C_VEL
LIN {X 0,Y 104.214,Z 823.764,A -85,B 0,C 180,E1 -26756.525,E2 -26756.525} C_VEL
LIN {X 0,Y 105.602,Z 822.532,A -85,B 0,C 180,E1 -26759.593,E2 -26759.593} C_VEL
LIN {X 0,Y 106.812,Z 819.991,A -85,B 0,C 180,E1 -26764.736,E2 -26764.736} C_VEL
LIN {X 0,Y 108.822,Z 816.755,A -85,B 0,C 180,E1 -26769.597,E2 -26769.597} C_VEL
LIN {X 0,Y 111.343,Z 814.419,A -85,B 0,C 180,E1 -26772.091,E2 -26772.091} C_VEL
LIN {X 0,Y 118.557,Z 808.571,A -85,B 0,C 180,E1 -26776.565,E2 -26776.565} C_VEL
LIN {X 0,Y 125.831,Z 801.822,A -85,B 0,C 180,E1 -26780.171,E2 -26780.171} C_VEL
LIN {X 0,Y 133.658,Z 793.488,A -85,B 0,C 180,E1 -26783.308,E2 -26783.308} C_VEL
LIN {X 0,Y 140.497,Z 784.926,A -85,B 0,C 180,E1 -26785.624,E2 -26785.624} C_VEL
LIN {X 0,Y 146.889,Z 775.571,A -85,B 0,C 180,E1 -26787.486,E2 -26787.486} C_VEL
LIN {X 0,Y 153.462,Z 764.015,A -85,B 0,C 180,E1 -26789.166,E2 -26789.166} C_VEL
LIN {X 0,Y 158.703,Z 752.486,A -85,B 0,C 180,E1 -26790.349,E2 -26790.349} C_VEL
LIN {X 0,Y 162.977,Z 740.125,A -85,B 0,C 180,E1 -26791.286,E2 -26791.286} C_VEL
LIN {X 0,Y 166.08,Z 727.649,A -85,B 0,C 180,E1 -26791.946,E2 -26791.946} C_VEL
LIN {X 0,Y 168.05,Z 714.071,A -85,B 0,C 180,E1 -26792.442,E2 -26792.442} C_VEL
LIN {X 0,Y 168.862,Z 705.269,A -85,B 0,C 180,E1 -26792.754,E2 -26792.754} C_VEL
LIN {X 0,Y 167.182,Z 701.095,A -85,B 0,C 180,E1 -26794.726,E2 -26794.726} C_VEL
LIN {X 0,Y 164.518,Z 695.762,A -85,B 0,C 180,E1 -26798.215,E2 -26798.215} C_VEL
LIN {X 0,Y 162.886,Z 692.593,A -85,B 0,C 180,E1 -26800.844,E2 -26800.844} C_VEL
LIN {X 0,Y 161.331,Z 689.55,A -85,B 0,C 180,E1 -26804.029,E2 -26804.029} C_VEL
LIN {X 0,Y 159.752,Z 685.881,A -85,B 0,C 180,E1 -26809.224,E2 -26809.224} C_VEL
LIN {X 0,Y 159.113,Z 685.385,A -85,B 0,C 180,E1 -26814.932,E2 -26814.932} C_VEL
LIN {X 0,Y 159.702,Z 685.532,A -85,B 0,C 180,E1 -26819.37,E2 -26819.37} C_VEL
LIN {X 0,Y 159.941,Z 686.031,A -85,B 0,C 180,E1 -26820.472,E2 -26820.472} C_VEL
LIN {X 0,Y 161.753,Z 690.034,A -85,B 0,C 180,E1 -26825.788,E2 -26825.788} C_VEL
LIN {X 0,Y 163.751,Z 694.154,A -85,B 0,C 180,E1 -26829.534,E2 -26829.534} C_VEL
LIN {X 0,Y 165.896,Z 698.4,A -85,B 0,C 180,E1 -26832.617,E2 -26832.617} C_VEL
LIN {X 0,Y 168.718,Z 704.472,A -85,B 0,C 180,E1 -26835.995,E2 -26835.995} C_VEL
LIN {X 0,Y 169.131,Z 705.43,A -85,B 0,C 180,E1 -26836.454,E2 -26836.454} C_VEL
LIN {X 0,Y 167.023,Z 718.966,A -85,B 0,C 180,E1 -26837.13,E2 -26837.13} C_VEL
LIN {X 0,Y 163.926,Z 731.297,A -85,B 0,C 180,E1 -26838.01,E2 -26838.01} C_VEL
LIN {X 0,Y 159.983,Z 742.813,A -85,B 0,C 180,E1 -26839.185,E2 -26839.185} C_VEL
LIN {X 0,Y 154.95,Z 754.069,A -85,B 0,C 180,E1 -26840.701,E2 -26840.701} C_VEL
LIN {X 0,Y 149.309,Z 764.362,A -85,B 0,C 180,E1 -26842.568,E2 -26842.568} C_VEL
LIN {X 0,Y 143.096,Z 773.623,A -85,B 0,C 180,E1 -26844.69,E2 -26844.69} C_VEL
LIN {X 0,Y 136.411,Z 782.021,A -85,B 0,C 180,E1 -26847.289,E2 -26847.289} C_VEL
LIN {X 0,Y 128.8,Z 790.137,A -85,B 0,C 180,E1 -26850.753,E2 -26850.753} C_VEL
LIN {X 0,Y 122.816,Z 795.603,A -85,B 0,C 180,E1 -26853.929,E2 -26853.929} C_VEL
LIN {X 0,Y 116.094,Z 800.875,A -85,B 0,C 180,E1 -26858.098,E2 -26858.098} C_VEL
LIN {X 0,Y 110.011,Z 804.902,A -85,B 0,C 180,E1 -26862.722,E2 -26862.722} C_VEL
LIN {X 0,Y 104.653,Z 807.819,A -85,B 0,C 180,E1 -26867.814,E2 -26867.814} C_VEL
LIN {X 0,Y 101.548,Z 809.189,A -85,B 0,C 180,E1 -26871.475,E2 -26871.475} C_VEL
LIN {X 0,Y 96.604,Z 810.648,A -85,B 0,C 180,E1 -26879.387,E2 -26879.387} C_VEL
LIN {X 0,Y 94.802,Z 810.759,A -85,B 0,C 180,E1 -26883.59,E2 -26883.59} C_VEL
LIN {X 0,Y 92.461,Z 809.72,A -85,B 0,C 180,E1 -26892.3,E2 -26892.3} C_VEL
LIN {X 0,Y 91.992,Z 808.611,A -85,B 0,C 180,E1 -26896.751,E2 -26896.751} C_VEL
LIN {X 0,Y 92.104,Z 806.412,A -85,B 0,C 180,E1 -26902.736,E2 -26902.736} C_VEL
LIN {X 0,Y 93.275,Z 802.64,A -85,B 0,C 180,E1 -26910,E2 -26910} C_VEL
LIN {X 0,Y 95.205,Z 798.081,A -85,B 0,C 180,E1 -26916.357,E2 -26916.357} C_VEL
LIN {X 0,Y 98.073,Z 792.281,A -85,B 0,C 180,E1 -26922.414,E2 -26922.414} C_VEL
LIN {X 0,Y 101.738,Z 785.058,A -85,B 0,C 180,E1 -26928.111,E2 -26928.111} C_VEL
LIN {X 0,Y 97.764,Z 782.704,A -85,B 0,C 180,E1 -26931.561,E2 -26931.561} C_VEL
LIN {X 0,Y 97.538,Z 782.469,A -85,B 0,C 180,E1 -26931.919,E2 -26931.919} C_VEL
LIN {X 0,Y 95.045,Z 789.825,A -85,B 0,C 180,E1 -26937.461,E2 -26937.461} C_VEL
LIN {X 0,Y 93.065,Z 796.425,A -85,B 0,C 180,E1 -26943.83,E2 -26943.83} C_VEL
LIN {X 0,Y 91.96,Z 801.567,A -85,B 0,C 180,E1 -26950.16,E2 -26950.16} C_VEL
LIN {X 0,Y 91.758,Z 805.554,A -85,B 0,C 180,E1 -26956.422,E2 -26956.422} C_VEL
LIN {X 0,Y 92.444,Z 808.566,A -85,B 0,C 180,E1 -26962.541,E2 -26962.541} C_VEL
LIN {X 0,Y 94.001,Z 810.738,A -85,B 0,C 180,E1 -26968.442,E2 -26968.442} C_VEL
LIN {X 0,Y 96.423,Z 812.182,A -85,B 0,C 180,E1 -26974.067,E2 -26974.067} C_VEL
LIN {X 0,Y 99.636,Z 812.912,A -85,B 0,C 180,E1 -26979.348,E2 -26979.348} C_VEL
LIN {X 0,Y 103.545,Z 812.918,A -85,B 0,C 180,E1 -26984.247,E2 -26984.247} C_VEL
LIN {X 0,Y 108.098,Z 812.289,A -85,B 0,C 180,E1 -26988.753,E2 -26988.753} C_VEL
LIN {X 0,Y 116.03,Z 810.005,A -85,B 0,C 180,E1 -26994.808,E2 -26994.808} C_VEL
LIN {X 0,Y 124.968,Z 806.163,A -85,B 0,C 180,E1 -27000,E2 -27000} C_VEL
LIN {X 0,Y 133.866,Z 801.127,A -85,B 0,C 180,E1 -27004.071,E2 -27004.071} C_VEL
LIN {X 0,Y 143.506,Z 794.343,A -85,B 0,C 180,E1 -27007.7,E2 -27007.7} C_VEL
LIN {X 0,Y 152.853,Z 786.189,A -85,B 0,C 180,E1 -27010.598,E2 -27010.598} C_VEL
LIN {X 0,Y 161.385,Z 777.273,A -85,B 0,C 180,E1 -27012.888,E2 -27012.888} C_VEL
LIN {X 0,Y 169.139,Z 767.37,A -85,B 0,C 180,E1 -27014.745,E2 -27014.745} C_VEL
LIN {X 0,Y 175.866,Z 756.909,A -85,B 0,C 180,E1 -27016.244,E2 -27016.244} C_VEL
LIN {X 0,Y 181.703,Z 745.726,A -85,B 0,C 180,E1 -27017.443,E2 -27017.443} C_VEL
LIN {X 0,Y 186.68,Z 733.492,A -85,B 0,C 180,E1 -27018.455,E2 -27018.455} C_VEL
LIN {X 0,Y 190.397,Z 721.148,A -85,B 0,C 180,E1 -27019.265,E2 -27019.265} C_VEL
LIN {X 0,Y 190.031,Z 721.465,A -85,B 0,C 180,E1 -27022.076,E2 -27022.076} C_VEL
LIN {X 0,Y 189.748,Z 724.435,A -85,B 0,C 180,E1 -27025.371,E2 -27025.371} C_VEL
LIN {X 0,Y 189.711,Z 724.729,A -85,B 0,C 180,E1 -27025.536,E2 -27025.536} C_VEL
LIN {X 0,Y 185.519,Z 738.057,A -85,B 0,C 180,E1 -27026.061,E2 -27026.061} C_VEL
LIN {X 0,Y 180.119,Z 750.837,A -85,B 0,C 180,E1 -27026.807,E2 -27026.807} C_VEL
LIN {X 0,Y 173.689,Z 762.803,A -85,B 0,C 180,E1 -27027.735,E2 -27027.735} C_VEL
LIN {X 0,Y 166.561,Z 773.613,A -85,B 0,C 180,E1 -27028.893,E2 -27028.893} C_VEL
LIN {X 0,Y 158.815,Z 783.39,A -85,B 0,C 180,E1 -27030.356,E2 -27030.356} C_VEL
LIN {X 0,Y 149.79,Z 793.017,A -85,B 0,C 180,E1 -27032.379,E2 -27032.379} C_VEL
LIN {X 0,Y 141.088,Z 800.955,A -85,B 0,C 180,E1 -27034.725,E2 -27034.725} C_VEL
LIN {X 0,Y 132.85,Z 807.431,A -85,B 0,C 180,E1 -27037.486,E2 -27037.486} C_VEL
LIN {X 0,Y 124.971,Z 812.731,A -85,B 0,C 180,E1 -27040.608,E2 -27040.608} C_VEL
LIN {X 0,Y 117.694,Z 817.004,A -85,B 0,C 180,E1 -27044.23,E2 -27044.23} C_VEL
LIN {X 0,Y 113.199,Z 819.351,A -85,B 0,C 180,E1 -27046.928,E2 -27046.928} C_VEL
LIN {X 0,Y 105.305,Z 822.832,A -85,B 0,C 180,E1 -27053.084,E2 -27053.084} C_VEL
LIN {X 0,Y 98.916,Z 824.896,A -85,B 0,C 180,E1 -27060.176,E2 -27060.176} C_VEL
LIN {X 0,Y 94.435,Z 825.558,A -85,B 0,C 180,E1 -27068.155,E2 -27068.155} C_VEL
LIN {X 0,Y 92.251,Z 824.799,A -85,B 0,C 180,E1 -27076.789,E2 -27076.789} C_VEL
LIN {X 0,Y 92.321,Z 822.514,A -85,B 0,C 180,E1 -27085.908,E2 -27085.908} C_VEL
LIN {X 0,Y 92.443,Z 823.839,A -85,B 0,C 180,E1 -27090,E2 -27090} C_VEL
LIN {X 0,Y 91.839,Z 825.134,A -85,B 0,C 180,E1 -27095.825,E2 -27095.825} C_VEL
LIN {X 0,Y 92.082,Z 825.738,A -85,B 0,C 180,E1 -27103.236,E2 -27103.236} C_VEL
LIN {X 0,Y 94.372,Z 825.055,A -85,B 0,C 180,E1 -27111.86,E2 -27111.86} C_VEL
LIN {X 0,Y 98.858,Z 822.776,A -85,B 0,C 180,E1 -27119.843,E2 -27119.843} C_VEL
LIN {X 0,Y 105.089,Z 818.901,A -85,B 0,C 180,E1 -27127.004,E2 -27127.004} C_VEL
LIN {X 0,Y 111.343,Z 814.419,A -85,B 0,C 180,E1 -27132.091,E2 -27132.091} C_VEL
LIN {X 0,Y 114.068,Z 811.919,A -85,B 0,C 180,E1 -27134.43,E2 -27134.43} C_VEL
LIN {X 0,Y 117.437,Z 807.44,A -85,B 0,C 180,E1 -27138.494,E2 -27138.494} C_VEL
LIN {X 0,Y 121.143,Z 802.411,A -85,B 0,C 180,E1 -27142.183,E2 -27142.183} C_VEL
LIN {X 0,Y 124.251,Z 798.976,A -85,B 0,C 180,E1 -27143.886,E2 -27143.886} C_VEL
LIN {X 0,Y 132.332,Z 790.291,A -85,B 0,C 180,E1 -27146.767,E2 -27146.767} C_VEL
LIN {X 0,Y 139.474,Z 781.221,A -85,B 0,C 180,E1 -27148.936,E2 -27148.936} C_VEL
LIN {X 0,Y 146.197,Z 771.158,A -85,B 0,C 180,E1 -27150.608,E2 -27150.608} C_VEL
LIN {X 0,Y 152.24,Z 760.051,A -85,B 0,C 180,E1 -27151.99,E2 -27151.99} C_VEL
LIN {X 0,Y 156.87,Z 749.559,A -85,B 0,C 180,E1 -27152.924,E2 -27152.924} C_VEL
LIN {X 0,Y 161.134,Z 736.782,A -85,B 0,C 180,E1 -27153.794,E2 -27153.794} C_VEL
LIN {X 0,Y 164.102,Z 723.844,A -85,B 0,C 180,E1 -27154.369,E2 -27154.369} C_VEL
LIN {X 0,Y 165.972,Z 708.872,A -85,B 0,C 180,E1 -27154.898,E2 -27154.898} C_VEL
LIN {X 0,Y 164.081,Z 704.605,A -85,B 0,C 180,E1 -27157.409,E2 -27157.409} C_VEL
LIN {X 0,Y 161.777,Z 699.641,A -85,B 0,C 180,E1 -27161.149,E2 -27161.149} C_VEL
LIN {X 0,Y 160.128,Z 696.275,A -85,B 0,C 180,E1 -27164.732,E2 -27164.732} C_VEL
LIN {X 0,Y 158.744,Z 692.833,A -85,B 0,C 180,E1 -27169.8,E2 -27169.8} C_VEL
LIN {X 0,Y 158.476,Z 692.341,A -85,B 0,C 180,E1 -27177.458,E2 -27177.458} C_VEL
LIN {X 0,Y 158.914,Z 692.833,A -85,B 0,C 180,E1 -27179.842,E2 -27179.842} C_VEL
LIN {X 0,Y 160.552,Z 696.86,A -85,B 0,C 180,E1 -27185.18,E2 -27185.18} C_VEL
LIN {X 0,Y 162.384,Z 700.896,A -85,B 0,C 180,E1 -27188.87,E2 -27188.87} C_VEL
LIN {X 0,Y 164.571,Z 705.546,A -85,B 0,C 180,E1 -27192.226,E2 -27192.226} C_VEL
LIN {X 0,Y 166.062,Z 709.373,A -85,B 0,C 180,E1 -27194.347,E2 -27194.347} C_VEL
LIN {X 0,Y 163.679,Z 722.391,A -85,B 0,C 180,E1 -27195.009,E2 -27195.009} C_VEL
LIN {X 0,Y 159.952,Z 735.467,A -85,B 0,C 180,E1 -27196.029,E2 -27196.029} C_VEL
LIN {X 0,Y 155.505,Z 747.098,A -85,B 0,C 180,E1 -27197.31,E2 -27197.31} C_VEL
LIN {X 0,Y 150.333,Z 757.612,A -85,B 0,C 180,E1 -27198.799,E2 -27198.799} C_VEL
LIN {X 0,Y 144.33,Z 767.524,A -85,B 0,C 180,E1 -27200.65,E2 -27200.65} C_VEL
LIN {X 0,Y 137.379,Z 776.994,A -85,B 0,C 180,E1 -27202.954,E2 -27202.954} C_VEL
LIN {X 0,Y 129.935,Z 785.54,A -85,B 0,C 180,E1 -27205.827,E2 -27205.827} C_VEL
LIN {X 0,Y 122.644,Z 792.559,A -85,B 0,C 180,E1 -27209.089,E2 -27209.089} C_VEL
LIN {X 0,Y 114.135,Z 799.439,A -85,B 0,C 180,E1 -27213.655,E2 -27213.655} C_VEL
LIN {X 0,Y 107.288,Z 804.022,A -85,B 0,C 180,E1 -27218.182,E2 -27218.182} C_VEL
LIN {X 0,Y 103.172,Z 806.353,A -85,B 0,C 180,E1 -27221.471,E2 -27221.471} C_VEL
LIN {X 0,Y 99.281,Z 808.273,A -85,B 0,C 180,E1 -27225.064,E2 -27225.064} C_VEL
LIN {X 0,Y 95.958,Z 809.678,A -85,B 0,C 180,E1 -27228.765,E2 -27228.765} C_VEL
LIN {X 0,Y 92.952,Z 810.647,A -85,B 0,C 180,E1 -27232.781,E2 -27232.781} C_VEL
LIN {X 0,Y 88.368,Z 811.378,A -85,B 0,C 180,E1 -27241.499,E2 -27241.499} C_VEL
LIN {X 0,Y 86.717,Z 811.106,A -85,B 0,C 180,E1 -27246.095,E2 -27246.095} C_VEL
LIN {X 0,Y 84.969,Z 809.356,A -85,B 0,C 180,E1 -27255.633,E2 -27255.633} C_VEL
LIN {X 0,Y 85.014,Z 806.979,A -85,B 0,C 180,E1 -27262.762,E2 -27262.762} C_VEL
LIN {X 0,Y 86.11,Z 803.529,A -85,B 0,C 180,E1 -27270,E2 -27270} C_VEL
LIN {X 0,Y 88.13,Z 799.059,A -85,B 0,C 180,E1 -27276.87,E2 -27276.87} C_VEL
LIN {X 0,Y 91.7,Z 792.277,A -85,B 0,C 180,E1 -27284.423,E2 -27284.423} C_VEL
LIN {X 0,Y 93.616,Z 788.796,A -85,B 0,C 180,E1 -27287.475,E2 -27287.475} C_VEL
LIN {X 0,Y 93.977,Z 787.661,A -85,B 0,C 180,E1 -27288.503,E2 -27288.503} C_VEL
LIN {X 0,Y 90.636,Z 785.968,A -85,B 0,C 180,E1 -27291.488,E2 -27291.488} C_VEL
LIN {X 0,Y 89.732,Z 785.197,A -85,B 0,C 180,E1 -27292.814,E2 -27292.814} C_VEL
LIN {X 0,Y 87.264,Z 792.193,A -85,B 0,C 180,E1 -27298.895,E2 -27298.895} C_VEL
LIN {X 0,Y 85.337,Z 799.101,A -85,B 0,C 180,E1 -27306.66,E2 -27306.66} C_VEL
LIN {X 0,Y 84.628,Z 804.584,A -85,B 0,C 180,E1 -27314.897,E2 -27314.897} C_VEL
LIN {X 0,Y 85.176,Z 808.103,A -85,B 0,C 180,E1 -27321.772,E2 -27321.772} C_VEL
LIN {X 0,Y 86.676,Z 810.624,A -85,B 0,C 180,E1 -27328.194,E2 -27328.194} C_VEL
LIN {X 0,Y 90.7,Z 812.948,A -85,B 0,C 180,E1 -27337.205,E2 -27337.205} C_VEL
LIN {X 0,Y 95.19,Z 813.673,A -85,B 0,C 180,E1 -27343.696,E2 -27343.696} C_VEL
LIN {X 0,Y 100.217,Z 813.496,A -85,B 0,C 180,E1 -27349.042,E2 -27349.042} C_VEL
LIN {X 0,Y 106.022,Z 812.477,A -85,B 0,C 180,E1 -27353.877,E2 -27353.877} C_VEL
LIN {X 0,Y 112.501,Z 810.616,A -85,B 0,C 180,E1 -27358.199,E2 -27358.199} C_VEL
LIN {X 0,Y 122.173,Z 806.693,A -85,B 0,C 180,E1 -27363.298,E2 -27363.298} C_VEL
LIN {X 0,Y 129.163,Z 803.061,A -85,B 0,C 180,E1 -27366.248,E2 -27366.248} C_VEL
LIN {X 0,Y 138.206,Z 797.314,A -85,B 0,C 180,E1 -27369.514,E2 -27369.514} C_VEL
LIN {X 0,Y 147.774,Z 789.909,A -85,B 0,C 180,E1 -27372.358,E2 -27372.358} C_VEL
LIN {X 0,Y 156.606,Z 781.616,A -85,B 0,C 180,E1 -27374.626,E2 -27374.626} C_VEL
LIN {X 0,Y 164.876,Z 772.12,A -85,B 0,C 180,E1 -27376.51,E2 -27376.51} C_VEL
LIN {X 0,Y 172.573,Z 761.494,A -85,B 0,C 180,E1 -27378.071,E2 -27378.071} C_VEL
LIN {X 0,Y 178.631,Z 751.204,A -85,B 0,C 180,E1 -27379.227,E2 -27379.227} C_VEL
LIN {X 0,Y 184.099,Z 739.462,A -85,B 0,C 180,E1 -27380.241,E2 -27380.241} C_VEL
LIN {X 0,Y 188.173,Z 728.08,A -85,B 0,C 180,E1 -27381.069,E2 -27381.069} C_VEL
LIN {X 0,Y 188.079,Z 728.287,A -85,B 0,C 180,E1 -27381.942,E2 -27381.942} C_VEL
LIN {X 0,Y 187.874,Z 729.326,A -85,B 0,C 180,E1 -27383.129,E2 -27383.129} C_VEL
LIN {X 0,Y 187.365,Z 731.164,A -85,B 0,C 180,E1 -27383.608,E2 -27383.608} C_VEL
LIN {X 0,Y 182.447,Z 744.104,A -85,B 0,C 180,E1 -27384.149,E2 -27384.149} C_VEL
LIN {X 0,Y 176.289,Z 756.539,A -85,B 0,C 180,E1 -27384.915,E2 -27384.915} C_VEL
LIN {X 0,Y 168.925,Z 768.385,A -85,B 0,C 180,E1 -27385.885,E2 -27385.885} C_VEL
LIN {X 0,Y 160.123,Z 779.926,A -85,B 0,C 180,E1 -27387.28,E2 -27387.28} C_VEL
LIN {X 0,Y 152.311,Z 788.53,A -85,B 0,C 180,E1 -27388.755,E2 -27388.755} C_VEL
LIN {X 0,Y 143.121,Z 797.103,A -85,B 0,C 180,E1 -27390.76,E2 -27390.76} C_VEL
LIN {X 0,Y 134.328,Z 804.078,A -85,B 0,C 180,E1 -27393.165,E2 -27393.165} C_VEL
LIN {X 0,Y 125.913,Z 809.859,A -85,B 0,C 180,E1 -27395.971,E2 -27395.971} C_VEL
LIN {X 0,Y 117.871,Z 814.566,A -85,B 0,C 180,E1 -27399.186,E2 -27399.186} C_VEL
LIN {X 0,Y 108.118,Z 819.298,A -85,B 0,C 180,E1 -27404.356,E2 -27404.356} C_VEL
LIN {X 0,Y 99.697,Z 822.562,A -85,B 0,C 180,E1 -27410.623,E2 -27410.623} C_VEL
LIN {X 0,Y 92.797,Z 824.374,A -85,B 0,C 180,E1 -27417.985,E2 -27417.985} C_VEL
LIN {X 0,Y 87.87,Z 824.782,A -85,B 0,C 180,E1 -27426.428,E2 -27426.428} C_VEL
LIN {X 0,Y 85.361,Z 823.833,A -85,B 0,C 180,E1 -27435.7,E2 -27435.7} C_VEL
LIN {X 0,Y 85.25,Z 821.481,A -85,B 0,C 180,E1 -27445.271,E2 -27445.271} C_VEL
LIN {X 0,Y 85.362,Z 823.099,A -85,B 0,C 180,E1 -27450,E2 -27450} C_VEL
LIN {X 0,Y 84.775,Z 824.385,A -85,B 0,C 180,E1 -27455.83,E2 -27455.83} C_VEL
LIN {X 0,Y 85.146,Z 825.114,A -85,B 0,C 180,E1 -27464.336,E2 -27464.336} C_VEL
LIN {X 0,Y 87.782,Z 824.493,A -85,B 0,C 180,E1 -27473.597,E2 -27473.597} C_VEL
LIN {X 0,Y 90.027,Z 823.617,A -85,B 0,C 180,E1 -27477.929,E2 -27477.929} C_VEL
LIN {X 0,Y 95.897,Z 820.61,A -85,B 0,C 180,E1 -27485.893,E2 -27485.893} C_VEL
LIN {X 0,Y 101.426,Z 817.266,A -85,B 0,C 180,E1 -27491.167,E2 -27491.167} C_VEL
LIN {X 0,Y 107.886,Z 812.888,A -85,B 0,C 180,E1 -27495.771,E2 -27495.771} C_VEL
LIN {X 0,Y 116.27,Z 806.32,A -85,B 0,C 180,E1 -27500.413,E2 -27500.413} C_VEL
LIN {X 0,Y 124.251,Z 798.976,A -85,B 0,C 180,E1 -27503.886,E2 -27503.886} C_VEL
LIN {X 0,Y 127.41,Z 795.375,A -85,B 0,C 180,E1 -27505.444,E2 -27505.444} C_VEL
LIN {X 0,Y 131.536,Z 789.15,A -85,B 0,C 180,E1 -27508.326,E2 -27508.326} C_VEL
LIN {X 0,Y 135.556,Z 782.462,A -85,B 0,C 180,E1 -27510.938,E2 -27510.938} C_VEL
LIN {X 0,Y 138.441,Z 778.055,A -85,B 0,C 180,E1 -27512.067,E2 -27512.067} C_VEL
LIN {X 0,Y 145.149,Z 767.755,A -85,B 0,C 180,E1 -27513.602,E2 -27513.602} C_VEL
LIN {X 0,Y 150.618,Z 757.578,A -85,B 0,C 180,E1 -27514.694,E2 -27514.694} C_VEL
LIN {X 0,Y 155.683,Z 745.588,A -85,B 0,C 180,E1 -27515.641,E2 -27515.641} C_VEL
LIN {X 0,Y 159.856,Z 732.161,A -85,B 0,C 180,E1 -27516.409,E2 -27516.409} C_VEL
LIN {X 0,Y 162.46,Z 719.353,A -85,B 0,C 180,E1 -27516.886,E2 -27516.886} C_VEL
LIN {X 0,Y 163.264,Z 712.885,A -85,B 0,C 180,E1 -27517.114,E2 -27517.114} C_VEL
LIN {X 0,Y 161.196,Z 708.159,A -85,B 0,C 180,E1 -27520.417,E2 -27520.417} C_VEL
LIN {X 0,Y 159.951,Z 705.335,A -85,B 0,C 180,E1 -27522.912,E2 -27522.912} C_VEL
LIN {X 0,Y 158.935,Z 703.008,A -85,B 0,C 180,E1 -27525.476,E2 -27525.476} C_VEL
LIN {X 0,Y 157.791,Z 699.829,A -85,B 0,C 180,E1 -27530.166,E2 -27530.166} C_VEL
LIN {X 0,Y 157.598,Z 699.388,A -85,B 0,C 180,E1 -27537.444,E2 -27537.444} C_VEL
LIN {X 0,Y 157.927,Z 699.78,A -85,B 0,C 180,E1 -27539.363,E2 -27539.363} C_VEL
LIN {X 0,Y 159.38,Z 703.697,A -85,B 0,C 180,E1 -27544.584,E2 -27544.584} C_VEL
LIN {X 0,Y 160.992,Z 707.596,A -85,B 0,C 180,E1 -27548.156,E2 -27548.156} C_VEL
LIN {X 0,Y 162.681,Z 711.888,A -85,B 0,C 180,E1 -27551.289,E2 -27551.289} C_VEL
LIN {X 0,Y 163.143,Z 713.559,A -85,B 0,C 180,E1 -27552.202,E2 -27552.202} C_VEL
LIN {X 0,Y 160.33,Z 726.495,A -85,B 0,C 180,E1 -27552.92,E2 -27552.92} C_VEL
LIN {X 0,Y 156.533,Z 738.488,A -85,B 0,C 180,E1 -27553.858,E2 -27553.858} C_VEL
LIN {X 0,Y 151.951,Z 749.494,A -85,B 0,C 180,E1 -27555.098,E2 -27555.098} C_VEL
LIN {X 0,Y 146.627,Z 759.627,A -85,B 0,C 180,E1 -27556.544,E2 -27556.544} C_VEL
LIN {X 0,Y 139.875,Z 770.087,A -85,B 0,C 180,E1 -27558.496,E2 -27558.496} C_VEL
LIN {X 0,Y 133.246,Z 778.573,A -85,B 0,C 180,E1 -27560.579,E2 -27560.579} C_VEL
LIN {X 0,Y 125.278,Z 787.123,A -85,B 0,C 180,E1 -27563.495,E2 -27563.495} C_VEL
LIN {X 0,Y 116.595,Z 794.883,A -85,B 0,C 180,E1 -27567.244,E2 -27567.244} C_VEL
LIN {X 0,Y 109.608,Z 800.11,A -85,B 0,C 180,E1 -27570.861,E2 -27570.861} C_VEL
LIN {X 0,Y 102.934,Z 804.323,A -85,B 0,C 180,E1 -27574.985,E2 -27574.985} C_VEL
LIN {X 0,Y 98.488,Z 806.73,A -85,B 0,C 180,E1 -27578.286,E2 -27578.286} C_VEL
LIN {X 0,Y 93.674,Z 808.942,A -85,B 0,C 180,E1 -27582.473,E2 -27582.473} C_VEL
LIN {X 0,Y 87.258,Z 811.175,A -85,B 0,C 180,E1 -27589.885,E2 -27589.885} C_VEL
LIN {X 0,Y 82.035,Z 811.981,A -85,B 0,C 180,E1 -27599.069,E2 -27599.069} C_VEL
LIN {X 0,Y 80.15,Z 811.775,A -85,B 0,C 180,E1 -27603.997,E2 -27603.997} C_VEL
LIN {X 0,Y 78.001,Z 810.096,A -85,B 0,C 180,E1 -27614.318,E2 -27614.318} C_VEL
LIN {X 0,Y 77.921,Z 807.542,A -85,B 0,C 180,E1 -27622.809,E2 -27622.809} C_VEL
LIN {X 0,Y 78.931,Z 804.416,A -85,B 0,C 180,E1 -27630,E2 -27630} C_VEL
LIN {X 0,Y 81.069,Z 800.02,A -85,B 0,C 180,E1 -27637.472,E2 -27637.472} C_VEL
LIN {X 0,Y 84.26,Z 794.439,A -85,B 0,C 180,E1 -27644.491,E2 -27644.491} C_VEL
LIN {X 0,Y 86.151,Z 791.154,A -85,B 0,C 180,E1 -27647.813,E2 -27647.813} C_VEL
LIN {X 0,Y 85.988,Z 790.091,A -85,B 0,C 180,E1 -27649.082,E2 -27649.082} C_VEL
LIN {X 0,Y 82.201,Z 788.102,A -85,B 0,C 180,E1 -27653.152,E2 -27653.152} C_VEL
LIN {X 0,Y 81.865,Z 787.778,A -85,B 0,C 180,E1 -27653.883,E2 -27653.883} C_VEL
LIN {X 0,Y 79.658,Z 794.134,A -85,B 0,C 180,E1 -27660.232,E2 -27660.232} C_VEL
LIN {X 0,Y 78.095,Z 799.849,A -85,B 0,C 180,E1 -27667.454,E2 -27667.454} C_VEL
LIN {X 0,Y 77.57,Z 805.313,A -85,B 0,C 180,E1 -27676.452,E2 -27676.452} C_VEL
LIN {X 0,Y 78.399,Z 808.749,A -85,B 0,C 180,E1 -27683.782,E2 -27683.782} C_VEL
LIN {X 0,Y 80.362,Z 811.365,A -85,B 0,C 180,E1 -27690.988,E2 -27690.988} C_VEL
LIN {X 0,Y 85.249,Z 813.708,A -85,B 0,C 180,E1 -27700.745,E2 -27700.745} C_VEL
LIN {X 0,Y 89.498,Z 814.361,A -85,B 0,C 180,E1 -27706.374,E2 -27706.374} C_VEL
LIN {X 0,Y 94.483,Z 814.298,A -85,B 0,C 180,E1 -27711.444,E2 -27711.444} C_VEL
LIN {X 0,Y 100.068,Z 813.582,A -85,B 0,C 180,E1 -27715.973,E2 -27715.973} C_VEL
LIN {X 0,Y 109.491,Z 811.224,A -85,B 0,C 180,E1 -27721.841,E2 -27721.841} C_VEL
LIN {X 0,Y 120.356,Z 806.987,A -85,B 0,C 180,E1 -27726.946,E2 -27726.946} C_VEL
LIN {X 0,Y 128.435,Z 802.896,A -85,B 0,C 180,E1 -27729.956,E2 -27729.956} C_VEL
LIN {X 0,Y 137.71,Z 797.117,A -85,B 0,C 180,E1 -27732.867,E2 -27732.867} C_VEL
LIN {X 0,Y 146.445,Z 790.508,A -85,B 0,C 180,E1 -27735.182,E2 -27735.182} C_VEL
LIN {X 0,Y 155.472,Z 782.358,A -85,B 0,C 180,E1 -27737.246,E2 -27737.246} C_VEL
LIN {X 0,Y 163.388,Z 773.707,A -85,B 0,C 180,E1 -27738.864,E2 -27738.864} C_VEL
LIN {X 0,Y 171.735,Z 762.571,A -85,B 0,C 180,E1 -27740.407,E2 -27740.407} C_VEL
LIN {X 0,Y 178.226,Z 751.83,A -85,B 0,C 180,E1 -27741.515,E2 -27741.515} C_VEL
LIN {X 0,Y 179.714,Z 748.958,A -85,B 0,C 180,E1 -27741.776,E2 -27741.776} C_VEL
LIN {X 0,Y 178.989,Z 750.494,A -85,B 0,C 180,E1 -27742.235,E2 -27742.235} C_VEL
LIN {X 0,Y 172.649,Z 761.654,A -85,B 0,C 180,E1 -27742.932,E2 -27742.932} C_VEL
LIN {X 0,Y 165.194,Z 772.352,A -85,B 0,C 180,E1 -27743.841,E2 -27743.841} C_VEL
LIN {X 0,Y 157.046,Z 782.057,A -85,B 0,C 180,E1 -27745.016,E2 -27745.016} C_VEL
LIN {X 0,Y 147.491,Z 791.594,A -85,B 0,C 180,E1 -27746.693,E2 -27746.693} C_VEL
LIN {X 0,Y 138.121,Z 799.494,A -85,B 0,C 180,E1 -27748.633,E2 -27748.633} C_VEL
LIN {X 0,Y 127.665,Z 806.857,A -85,B 0,C 180,E1 -27751.432,E2 -27751.432} C_VEL
LIN {X 0,Y 116.255,Z 813.437,A -85,B 0,C 180,E1 -27755.304,E2 -27755.304} C_VEL
LIN {X 0,Y 108.272,Z 817.231,A -85,B 0,C 180,E1 -27758.839,E2 -27758.839} C_VEL
LIN {X 0,Y 98.593,Z 820.943,A -85,B 0,C 180,E1 -27764.536,E2 -27764.536} C_VEL
LIN {X 0,Y 90.386,Z 823.186,A -85,B 0,C 180,E1 -27771.536,E2 -27771.536} C_VEL
LIN {X 0,Y 83.902,Z 824.072,A -85,B 0,C 180,E1 -27779.829,E2 -27779.829} C_VEL
LIN {X 0,Y 79.617,Z 823.599,A -85,B 0,C 180,E1 -27789.324,E2 -27789.324} C_VEL
LIN {X 0,Y 78.093,Z 821.699,A -85,B 0,C 180,E1 -27799.631,E2 -27799.631} C_VEL
LIN {X 0,Y 78.204,Z 820.491,A -85,B 0,C 180,E1 -27804.254,E2 -27804.254} C_VEL
LIN {X 0,Y 78.281,Z 822.356,A -85,B 0,C 180,E1 -27810,E2 -27810} C_VEL
LIN {X 0,Y 77.727,Z 823.619,A -85,B 0,C 180,E1 -27815.949,E2 -27815.949} C_VEL
LIN {X 0,Y 78.26,Z 824.491,A -85,B 0,C 180,E1 -27825.629,E2 -27825.629} C_VEL
LIN {X 0,Y 81.287,Z 823.932,A -85,B 0,C 180,E1 -27835.613,E2 -27835.613} C_VEL
LIN {X 0,Y 83.792,Z 823.1,A -85,B 0,C 180,E1 -27840.214,E2 -27840.214} C_VEL
LIN {X 0,Y 86.762,Z 821.843,A -85,B 0,C 180,E1 -27844.542,E2 -27844.542} C_VEL
LIN {X 0,Y 94.079,Z 818.108,A -85,B 0,C 180,E1 -27852.246,E2 -27852.246} C_VEL
LIN {X 0,Y 100.678,Z 814.159,A -85,B 0,C 180,E1 -27857.135,E2 -27857.135} C_VEL
LIN {X 0,Y 107.993,Z 809.103,A -85,B 0,C 180,E1 -27861.345,E2 -27861.345} C_VEL
LIN {X 0,Y 115.881,Z 802.791,A -85,B 0,C 180,E1 -27864.958,E2 -27864.958} C_VEL
LIN {X 0,Y 124.254,Z 794.931,A -85,B 0,C 180,E1 -27868.039,E2 -27868.039} C_VEL
LIN {X 0,Y 133.013,Z 785.185,A -85,B 0,C 180,E1 -27870.667,E2 -27870.667} C_VEL
LIN {X 0,Y 138.441,Z 778.055,A -85,B 0,C 180,E1 -27872.067,E2 -27872.067} C_VEL
LIN {X 0,Y 141.244,Z 773.496,A -85,B 0,C 180,E1 -27873.108,E2 -27873.108} C_VEL
LIN {X 0,Y 144.861,Z 765.82,A -85,B 0,C 180,E1 -27875.171,E2 -27875.171} C_VEL
LIN {X 0,Y 148.185,Z 757.769,A -85,B 0,C 180,E1 -27876.978,E2 -27876.978} C_VEL
LIN {X 0,Y 150.435,Z 752.574,A -85,B 0,C 180,E1 -27877.628,E2 -27877.628} C_VEL
LIN {X 0,Y 154.93,Z 741.166,A -85,B 0,C 180,E1 -27878.397,E2 -27878.397} C_VEL
LIN {X 0,Y 158.654,Z 728.153,A -85,B 0,C 180,E1 -27878.981,E2 -27878.981} C_VEL
LIN {X 0,Y 160.653,Z 717.155,A -85,B 0,C 180,E1 -27879.431,E2 -27879.431} C_VEL
LIN {X 0,Y 159.048,Z 712.793,A -85,B 0,C 180,E1 -27882.812,E2 -27882.812} C_VEL
LIN {X 0,Y 157.799,Z 709.764,A -85,B 0,C 180,E1 -27886.149,E2 -27886.149} C_VEL
LIN {X 0,Y 156.847,Z 706.813,A -85,B 0,C 180,E1 -27890.538,E2 -27890.538} C_VEL
LIN {X 0,Y 156.934,Z 706.583,A -85,B 0,C 180,E1 -27898.717,E2 -27898.717} C_VEL
LIN {X 0,Y 158.09,Z 710.359,A -85,B 0,C 180,E1 -27903.824,E2 -27903.824} C_VEL
LIN {X 0,Y 159.311,Z 714.077,A -85,B 0,C 180,E1 -27907.286,E2 -27907.286} C_VEL
LIN {X 0,Y 160.396,Z 717.507,A -85,B 0,C 180,E1 -27909.935,E2 -27909.935} C_VEL
LIN {X 0,Y 157.347,Z 729.892,A -85,B 0,C 180,E1 -27910.699,E2 -27910.699} C_VEL
LIN {X 0,Y 152.988,Z 742.215,A -85,B 0,C 180,E1 -27911.702,E2 -27911.702} C_VEL
LIN {X 0,Y 147.86,Z 753.411,A -85,B 0,C 180,E1 -27913,E2 -27913} C_VEL
LIN {X 0,Y 141.756,Z 763.888,A -85,B 0,C 180,E1 -27914.554,E2 -27914.554} C_VEL
LIN {X 0,Y 133.897,Z 774.752,A -85,B 0,C 180,E1 -27916.687,E2 -27916.687} C_VEL
LIN {X 0,Y 126.388,Z 783.316,A -85,B 0,C 180,E1 -27919.041,E2 -27919.041} C_VEL
LIN {X 0,Y 117.664,Z 791.528,A -85,B 0,C 180,E1 -27922.214,E2 -27922.214} C_VEL
LIN {X 0,Y 109.331,Z 798.075,A -85,B 0,C 180,E1 -27925.852,E2 -27925.852} C_VEL
LIN {X 0,Y 101.444,Z 803.212,A -85,B 0,C 180,E1 -27930.006,E2 -27930.006} C_VEL
LIN {X 0,Y 94.135,Z 807.106,A -85,B 0,C 180,E1 -27934.793,E2 -27934.793} C_VEL
LIN {X 0,Y 88.319,Z 809.599,A -85,B 0,C 180,E1 -27939.539,E2 -27939.539} C_VEL
LIN {X 0,Y 81.808,Z 811.702,A -85,B 0,C 180,E1 -27946.587,E2 -27946.587} C_VEL
LIN {X 0,Y 75.876,Z 812.582,A -85,B 0,C 180,E1 -27956.239,E2 -27956.239} C_VEL
LIN {X 0,Y 73.71,Z 812.43,A -85,B 0,C 180,E1 -27961.529,E2 -27961.529} C_VEL
LIN {X 0,Y 72.05,Z 811.84,A -85,B 0,C 180,E1 -27967.035,E2 -27967.035} C_VEL
LIN {X 0,Y 71.063,Z 810.838,A -85,B 0,C 180,E1 -27972.741,E2 -27972.741} C_VEL
LIN {X 0,Y 70.846,Z 808.138,A -85,B 0,C 180,E1 -27982.752,E2 -27982.752} C_VEL
LIN {X 0,Y 72.407,Z 803.993,A -85,B 0,C 180,E1 -27992.782,E2 -27992.782} C_VEL
LIN {X 0,Y 74.982,Z 799.298,A -85,B 0,C 180,E1 -28000.804,E2 -28000.804} C_VEL
LIN {X 0,Y 78.718,Z 793.361,A -85,B 0,C 180,E1 -28008.208,E2 -28008.208} C_VEL
LIN {X 0,Y 75.93,Z 791.434,A -85,B 0,C 180,E1 -28012.242,E2 -28012.242} C_VEL
LIN {X 0,Y 74.313,Z 790.572,A -85,B 0,C 180,E1 -28014.334,E2 -28014.334} C_VEL
LIN {X 0,Y 73.926,Z 790.304,A -85,B 0,C 180,E1 -28015.263,E2 -28015.263} C_VEL
LIN {X 0,Y 71.831,Z 796.566,A -85,B 0,C 180,E1 -28022.651,E2 -28022.651} C_VEL
LIN {X 0,Y 70.505,Z 802.983,A -85,B 0,C 180,E1 -28032.494,E2 -28032.494} C_VEL
LIN {X 0,Y 71.236,Z 808.365,A -85,B 0,C 180,E1 -28043.704,E2 -28043.704} C_VEL
LIN {X 0,Y 73.127,Z 811.163,A -85,B 0,C 180,E1 -28051.28,E2 -28051.28} C_VEL
LIN {X 0,Y 76.198,Z 813.204,A -85,B 0,C 180,E1 -28058.35,E2 -28058.35} C_VEL
LIN {X 0,Y 80.168,Z 814.464,A -85,B 0,C 180,E1 -28064.752,E2 -28064.752} C_VEL
LIN {X 0,Y 85.413,Z 815.086,A -85,B 0,C 180,E1 -28070.881,E2 -28070.881} C_VEL
LIN {X 0,Y 91.552,Z 814.938,A -85,B 0,C 180,E1 -28076.305,E2 -28076.305} C_VEL
LIN {X 0,Y 98.406,Z 813.957,A -85,B 0,C 180,E1 -28081.038,E2 -28081.038} C_VEL
LIN {X 0,Y 105.841,Z 812.163,A -85,B 0,C 180,E1 -28085.126,E2 -28085.126} C_VEL
LIN {X 0,Y 113.742,Z 809.527,A -85,B 0,C 180,E1 -28088.659,E2 -28088.659} C_VEL
LIN {X 0,Y 122.002,Z 805.985,A -85,B 0,C 180,E1 -28091.688,E2 -28091.688} C_VEL
LIN {X 0,Y 130.563,Z 801.439,A -85,B 0,C 180,E1 -28094.33,E2 -28094.33} C_VEL
LIN {X 0,Y 139.342,Z 795.832,A -85,B 0,C 180,E1 -28096.609,E2 -28096.609} C_VEL
LIN {X 0,Y 148.319,Z 788.907,A -85,B 0,C 180,E1 -28098.62,E2 -28098.62} C_VEL
LIN {X 0,Y 157.483,Z 780.362,A -85,B 0,C 180,E1 -28100.423,E2 -28100.423} C_VEL
LIN {X 0,Y 162.22,Z 775.238,A -85,B 0,C 180,E1 -28101.271,E2 -28101.271} C_VEL
LIN {X 0,Y 160.884,Z 776.859,A -85,B 0,C 180,E1 -28101.798,E2 -28101.798} C_VEL
LIN {X 0,Y 152.589,Z 785.732,A -85,B 0,C 180,E1 -28102.906,E2 -28102.906} C_VEL
LIN {X 0,Y 142.884,Z 794.468,A -85,B 0,C 180,E1 -28104.504,E2 -28104.504} C_VEL
LIN {X 0,Y 133.304,Z 801.668,A -85,B 0,C 180,E1 -28106.331,E2 -28106.331} C_VEL
LIN {X 0,Y 124.132,Z 807.554,A -85,B 0,C 180,E1 -28108.652,E2 -28108.652} C_VEL
LIN {X 0,Y 115.23,Z 812.369,A -85,B 0,C 180,E1 -28111.366,E2 -28111.366} C_VEL
LIN {X 0,Y 106.689,Z 816.21,A -85,B 0,C 180,E1 -28114.574,E2 -28114.574} C_VEL
LIN {X 0,Y 98.706,Z 819.176,A -85,B 0,C 180,E1 -28118.446,E2 -28118.446} C_VEL
LIN {X 0,Y 89.151,Z 821.88,A -85,B 0,C 180,E1 -28124.808,E2 -28124.808} C_VEL
LIN {X 0,Y 81.068,Z 823.214,A -85,B 0,C 180,E1 -28132.639,E2 -28132.639} C_VEL
LIN {X 0,Y 75.056,Z 823.15,A -85,B 0,C 180,E1 -28142.084,E2 -28142.084} C_VEL
LIN {X 0,Y 71.722,Z 821.746,A -85,B 0,C 180,E1 -28152.905,E2 -28152.905} C_VEL
LIN {X 0,Y 71.183,Z 819.46,A -85,B 0,C 180,E1 -28163.078,E2 -28163.078} C_VEL
LIN {X 0,Y 71.2,Z 821.613,A -85,B 0,C 180,E1 -28170,E2 -28170} C_VEL
LIN {X 0,Y 70.667,Z 822.811,A -85,B 0,C 180,E1 -28175.997,E2 -28175.997} C_VEL
LIN {X 0,Y 71.4,Z 823.865,A -85,B 0,C 180,E1 -28187.175,E2 -28187.175} C_VEL
LIN {X 0,Y 74.913,Z 823.37,A -85,B 0,C 180,E1 -28197.974,E2 -28197.974} C_VEL
LIN {X 0,Y 80.984,Z 821.375,A -85,B 0,C 180,E1 -28207.406,E2 -28207.406} C_VEL
LIN {X 0,Y 88.929,Z 817.708,A -85,B 0,C 180,E1 -28215.336,E2 -28215.336} C_VEL
LIN {X 0,Y 95.97,Z 813.83,A -85,B 0,C 180,E1 -28220.256,E2 -28220.256} C_VEL
LIN {X 0,Y 103.707,Z 808.851,A -85,B 0,C 180,E1 -28224.409,E2 -28224.409} C_VEL
LIN {X 0,Y 111.959,Z 802.626,A -85,B 0,C 180,E1 -28227.931,E2 -28227.931} C_VEL
LIN {X 0,Y 120.649,Z 794.905,A -85,B 0,C 180,E1 -28230.898,E2 -28230.898} C_VEL
LIN {X 0,Y 129.691,Z 785.276,A -85,B 0,C 180,E1 -28233.395,E2 -28233.395} C_VEL
LIN {X 0,Y 136.636,Z 776.42,A -85,B 0,C 180,E1 -28235.031,E2 -28235.031} C_VEL
LIN {X 0,Y 143.734,Z 765.537,A -85,B 0,C 180,E1 -28236.459,E2 -28236.459} C_VEL
LIN {X 0,Y 150.149,Z 753.201,A -85,B 0,C 180,E1 -28237.58,E2 -28237.58} C_VEL
LIN {X 0,Y 150.435,Z 752.574,A -85,B 0,C 180,E1 -28237.628,E2 -28237.628} C_VEL
LIN {X 0,Y 152.52,Z 747.289,A -85,B 0,C 180,E1 -28238.246,E2 -28238.246} C_VEL
LIN {X 0,Y 154.906,Z 738.586,A -85,B 0,C 180,E1 -28239.783,E2 -28239.783} C_VEL
LIN {X 0,Y 156.699,Z 729.624,A -85,B 0,C 180,E1 -28241.188,E2 -28241.188} C_VEL
LIN {X 0,Y 157.777,Z 723.939,A -85,B 0,C 180,E1 -28241.606,E2 -28241.606} C_VEL
LIN {X 0,Y 158.175,Z 721.562,A -85,B 0,C 180,E1 -28241.768,E2 -28241.768} C_VEL
LIN {X 0,Y 157.081,Z 718.141,A -85,B 0,C 180,E1 -28244.926,E2 -28244.926} C_VEL
LIN {X 0,Y 156.566,Z 716.593,A -85,B 0,C 180,E1 -28246.7,E2 -28246.7} C_VEL
LIN {X 0,Y 155.841,Z 713.832,A -85,B 0,C 180,E1 -28250.745,E2 -28250.745} C_VEL
LIN {X 0,Y 155.839,Z 713.599,A -85,B 0,C 180,E1 -28258.385,E2 -28258.385} C_VEL
LIN {X 0,Y 156.554,Z 716.958,A -85,B 0,C 180,E1 -28263.056,E2 -28263.056} C_VEL
LIN {X 0,Y 157.361,Z 720.464,A -85,B 0,C 180,E1 -28266.411,E2 -28266.411} C_VEL
LIN {X 0,Y 157.737,Z 721.881,A -85,B 0,C 180,E1 -28267.681,E2 -28267.681} C_VEL
LIN {X 0,Y 154.123,Z 734.571,A -85,B 0,C 180,E1 -28268.476,E2 -28268.476} C_VEL
LIN {X 0,Y 149.623,Z 745.957,A -85,B 0,C 180,E1 -28269.47,E2 -28269.47} C_VEL
LIN {X 0,Y 143.945,Z 757.072,A -85,B 0,C 180,E1 -28270.716,E2 -28270.716} C_VEL
LIN {X 0,Y 136.757,Z 768.337,A -85,B 0,C 180,E1 -28272.474,E2 -28272.474} C_VEL
LIN {X 0,Y 128.854,Z 778.204,A -85,B 0,C 180,E1 -28274.51,E2 -28274.51} C_VEL
LIN {X 0,Y 120.839,Z 786.513,A -85,B 0,C 180,E1 -28276.906,E2 -28276.906} C_VEL
LIN {X 0,Y 112.146,Z 793.995,A -85,B 0,C 180,E1 -28279.949,E2 -28279.949} C_VEL
LIN {X 0,Y 103.241,Z 800.299,A -85,B 0,C 180,E1 -28283.713,E2 -28283.713} C_VEL
LIN {X 0,Y 95.317,Z 804.912,A -85,B 0,C 180,E1 -28287.776,E2 -28287.776} C_VEL
LIN {X 0,Y 87.709,Z 808.516,A -85,B 0,C 180,E1 -28292.719,E2 -28292.719} C_VEL
LIN {X 0,Y 80.796,Z 811.053,A -85,B 0,C 180,E1 -28298.478,E2 -28298.478} C_VEL
LIN {X 0,Y 76.669,Z 812.209,A -85,B 0,C 180,E1 -28302.835,E2 -28302.835} C_VEL
LIN {X 0,Y 73.031,Z 812.907,A -85,B 0,C 180,E1 -28307.653,E2 -28307.653} C_VEL
LIN {X 0,Y 69.315,Z 813.2,A -85,B 0,C 180,E1 -28314.207,E2 -28314.207} C_VEL
LIN {X 0,Y 65.441,Z 812.546,A -85,B 0,C 180,E1 -28324.56,E2 -28324.56} C_VEL
LIN {X 0,Y 64.207,Z 811.578,A -85,B 0,C 180,E1 -28330.83,E2 -28330.83} C_VEL
LIN {X 0,Y 63.756,Z 808.704,A -85,B 0,C 180,E1 -28342.795,E2 -28342.795} C_VEL
LIN {X 0,Y 65.257,Z 804.916,A -85,B 0,C 180,E1 -28353.087,E2 -28353.087} C_VEL
LIN {X 0,Y 68.004,Z 800.302,A -85,B 0,C 180,E1 -28361.928,E2 -28361.928} C_VEL
LIN {X 0,Y 71.223,Z 795.497,A -85,B 0,C 180,E1 -28368.786,E2 -28368.786} C_VEL
LIN {X 0,Y 66.316,Z 792.857,A -85,B 0,C 180,E1 -28376.119,E2 -28376.119} C_VEL
LIN {X 0,Y 66.096,Z 792.591,A -85,B 0,C 180,E1 -28376.865,E2 -28376.865} C_VEL
LIN {X 0,Y 64.014,Z 799.145,A -85,B 0,C 180,E1 -28386.125,E2 -28386.125} C_VEL
LIN {X 0,Y 63.385,Z 804.058,A -85,B 0,C 180,E1 -28394.977,E2 -28394.977} C_VEL
LIN {X 0,Y 64.712,Z 809.256,A -85,B 0,C 180,E1 -28407.11,E2 -28407.11} C_VEL
LIN {X 0,Y 68.309,Z 812.731,A -85,B 0,C 180,E1 -28417.812,E2 -28417.812} C_VEL
LIN {X 0,Y 72.617,Z 814.538,A -85,B 0,C 180,E1 -28425.418,E2 -28425.418} C_VEL
LIN {X 0,Y 78.049,Z 815.568,A -85,B 0,C 180,E1 -28432.09,E2 -28432.09} C_VEL
LIN {X 0,Y 87.242,Z 815.705,A -85,B 0,C 180,E1 -28440,E2 -28440} C_VEL
LIN {X 0,Y 93.941,Z 814.929,A -85,B 0,C 180,E1 -28444.291,E2 -28444.291} C_VEL
LIN {X 0,Y 101.145,Z 813.504,A -85,B 0,C 180,E1 -28447.988,E2 -28447.988} C_VEL
LIN {X 0,Y 112.531,Z 809.991,A -85,B 0,C 180,E1 -28452.576,E2 -28452.576} C_VEL
LIN {X 0,Y 124.437,Z 804.869,A -85,B 0,C 180,E1 -28456.237,E2 -28456.237} C_VEL
LIN {X 0,Y 133.375,Z 799.934,A -85,B 0,C 180,E1 -28458.475,E2 -28458.475} C_VEL
LIN {X 0,Y 143.553,Z 792.994,A -85,B 0,C 180,E1 -28460.627,E2 -28460.627} C_VEL
LIN {X 0,Y 144.593,Z 792.203,A -85,B 0,C 180,E1 -28460.835,E2 -28460.835} C_VEL
LIN {X 0,Y 143.401,Z 793.243,A -85,B 0,C 180,E1 -28461.384,E2 -28461.384} C_VEL
LIN {X 0,Y 133.578,Z 800.529,A -85,B 0,C 180,E1 -28462.97,E2 -28462.97} C_VEL
LIN {X 0,Y 124.021,Z 806.475,A -85,B 0,C 180,E1 -28464.952,E2 -28464.952} C_VEL
LIN {X 0,Y 114.753,Z 811.313,A -85,B 0,C 180,E1 -28467.374,E2 -28467.374} C_VEL
LIN {X 0,Y 105.732,Z 815.223,A -85,B 0,C 180,E1 -28470.221,E2 -28470.221} C_VEL
LIN {X 0,Y 94.45,Z 819.08,A -85,B 0,C 180,E1 -28475.066,E2 -28475.066} C_VEL
LIN {X 0,Y 84.274,Z 821.497,A -85,B 0,C 180,E1 -28481.363,E2 -28481.363} C_VEL
LIN {X 0,Y 75.533,Z 822.538,A -85,B 0,C 180,E1 -28489.36,E2 -28489.36} C_VEL
LIN {X 0,Y 68.866,Z 822.259,A -85,B 0,C 180,E1 -28499.319,E2 -28499.319} C_VEL
LIN {X 0,Y 64.994,Z 820.652,A -85,B 0,C 180,E1 -28511.071,E2 -28511.071} C_VEL
LIN {X 0,Y 64.165,Z 818.417,A -85,B 0,C 180,E1 -28521.626,E2 -28521.626} C_VEL
LIN {X 0,Y 64.121,Z 820.869,A -85,B 0,C 180,E1 -28530,E2 -28530} C_VEL
LIN {X 0,Y 63.597,Z 822.046,A -85,B 0,C 180,E1 -28536.344,E2 -28536.344} C_VEL
LIN {X 0,Y 64.616,Z 823.224,A -85,B 0,C 180,E1 -28549.044,E2 -28549.044} C_VEL
LIN {X 0,Y 68.696,Z 822.809,A -85,B 0,C 180,E1 -28560.765,E2 -28560.765} C_VEL
LIN {X 0,Y 75.441,Z 820.89,A -85,B 0,C 180,E1 -28570.699,E2 -28570.699} C_VEL
LIN {X 0,Y 79.512,Z 819.306,A -85,B 0,C 180,E1 -28574.999,E2 -28574.999} C_VEL
LIN {X 0,Y 86.473,Z 816.169,A -85,B 0,C 180,E1 -28580.542,E2 -28580.542} C_VEL
LIN {X 0,Y 94.239,Z 812.014,A -85,B 0,C 180,E1 -28585.117,E2 -28585.117} C_VEL
LIN {X 0,Y 103.971,Z 805.692,A -85,B 0,C 180,E1 -28589.522,E2 -28589.522} C_VEL
LIN {X 0,Y 112.817,Z 798.861,A -85,B 0,C 180,E1 -28592.584,E2 -28592.584} C_VEL
LIN {X 0,Y 121.986,Z 790.385,A -85,B 0,C 180,E1 -28595.146,E2 -28595.146} C_VEL
LIN {X 0,Y 129.781,Z 781.709,A -85,B 0,C 180,E1 -28597.011,E2 -28597.011} C_VEL
LIN {X 0,Y 137.836,Z 771.058,A -85,B 0,C 180,E1 -28598.514,E2 -28598.514} C_VEL
LIN {X 0,Y 144.314,Z 760.427,A -85,B 0,C 180,E1 -28599.626,E2 -28599.626} C_VEL
LIN {X 0,Y 150.06,Z 748.544,A -85,B 0,C 180,E1 -28600.498,E2 -28600.498} C_VEL
LIN {X 0,Y 154.723,Z 735.807,A -85,B 0,C 180,E1 -28601.184,E2 -28601.184} C_VEL
LIN {X 0,Y 157.777,Z 723.939,A -85,B 0,C 180,E1 -28601.606,E2 -28601.606} C_VEL
LIN {X 0,Y 158.003,Z 721.772,A -85,B 0,C 180,E1 -28601.968,E2 -28601.968} C_VEL
LIN {X 0,Y 157.825,Z 719.766,A -85,B 0,C 180,E1 -28602.95,E2 -28602.95} C_VEL
LIN {X 0,Y 157.192,Z 718.53,A -85,B 0,C 180,E1 -28604.584,E2 -28604.584} C_VEL
LIN {X 0,Y 156.147,Z 718.648,A -85,B 0,C 180,E1 -28606.864,E2 -28606.864} C_VEL
LIN {X 0,Y 154.532,Z 720.339,A -85,B 0,C 180,E1 -28611.359,E2 -28611.359} C_VEL
LIN {X 0,Y 154.248,Z 720.568,A -85,B 0,C 180,E1 -28613.19,E2 -28613.19} C_VEL
LIN {X 0,Y 154.412,Z 720.594,A -85,B 0,C 180,E1 -28618.044,E2 -28618.044} C_VEL
LIN {X 0,Y 154.763,Z 723.781,A -85,B 0,C 180,E1 -28622.603,E2 -28622.603} C_VEL
LIN {X 0,Y 155.138,Z 726.55,A -85,B 0,C 180,E1 -28625.361,E2 -28625.361} C_VEL
LIN {X 0,Y 150.806,Z 739.638,A -85,B 0,C 180,E1 -28626.206,E2 -28626.206} C_VEL
LIN {X 0,Y 145.264,Z 751.873,A -85,B 0,C 180,E1 -28627.352,E2 -28627.352} C_VEL
LIN {X 0,Y 139.669,Z 761.6,A -85,B 0,C 180,E1 -28628.519,E2 -28628.519} C_VEL
LIN {X 0,Y 132.094,Z 772.282,A -85,B 0,C 180,E1 -28630.181,E2 -28630.181} C_VEL
LIN {X 0,Y 124.002,Z 781.512,A -85,B 0,C 180,E1 -28632.137,E2 -28632.137} C_VEL
LIN {X 0,Y 114.518,Z 790.377,A -85,B 0,C 180,E1 -28634.859,E2 -28634.859} C_VEL
LIN {X 0,Y 105.31,Z 797.413,A -85,B 0,C 180,E1 -28638.016,E2 -28638.016} C_VEL
LIN {X 0,Y 94.993,Z 803.73,A -85,B 0,C 180,E1 -28642.364,E2 -28642.364} C_VEL
LIN {X 0,Y 86.644,Z 807.802,A -85,B 0,C 180,E1 -28646.846,E2 -28646.846} C_VEL
LIN {X 0,Y 78.569,Z 810.875,A -85,B 0,C 180,E1 -28652.459,E2 -28652.459} C_VEL
LIN {X 0,Y 71.907,Z 812.701,A -85,B 0,C 180,E1 -28658.567,E2 -28658.567} C_VEL
LIN {X 0,Y 67.823,Z 813.471,A -85,B 0,C 180,E1 -28663.503,E2 -28663.503} C_VEL
LIN {X 0,Y 61.314,Z 813.704,A -85,B 0,C 180,E1 -28675.033,E2 -28675.033} C_VEL
LIN {X 0,Y 58.979,Z 813.237,A -85,B 0,C 180,E1 -28681.534,E2 -28681.534} C_VEL
LIN {X 0,Y 57.408,Z 812.321,A -85,B 0,C 180,E1 -28688.454,E2 -28688.454} C_VEL
LIN {X 0,Y 56.651,Z 810.991,A -85,B 0,C 180,E1 -28695.634,E2 -28695.634} C_VEL
LIN {X 0,Y 56.986,Z 808.206,A -85,B 0,C 180,E1 -28706.465,E2 -28706.465} C_VEL
LIN {X 0,Y 58.958,Z 804.407,A -85,B 0,C 180,E1 -28716.846,E2 -28716.846} C_VEL
LIN {X 0,Y 62.372,Z 799.5,A -85,B 0,C 180,E1 -28726.361,E2 -28726.361} C_VEL
LIN {X 0,Y 63.412,Z 797.65,A -85,B 0,C 180,E1 -28729.42,E2 -28729.42} C_VEL
LIN {X 0,Y 58.183,Z 794.939,A -85,B 0,C 180,E1 -28739.164,E2 -28739.164} C_VEL
LIN {X 0,Y 56.593,Z 800.456,A -85,B 0,C 180,E1 -28748.383,E2 -28748.383} C_VEL
LIN {X 0,Y 56.633,Z 806.585,A -85,B 0,C 180,E1 -28761.648,E2 -28761.648} C_VEL
LIN {X 0,Y 59.559,Z 811.245,A -85,B 0,C 180,E1 -28774.836,E2 -28774.836} C_VEL
LIN {X 0,Y 65.105,Z 814.406,A -85,B 0,C 180,E1 -28786.293,E2 -28786.293} C_VEL
LIN {X 0,Y 71.478,Z 815.959,A -85,B 0,C 180,E1 -28794.357,E2 -28794.357} C_VEL
LIN {X 0,Y 77.651,Z 816.514,A -85,B 0,C 180,E1 -28800,E2 -28800} C_VEL
LIN {X 0,Y 84.642,Z 816.41,A -85,B 0,C 180,E1 -28804.893,E2 -28804.893} C_VEL
LIN {X 0,Y 92.559,Z 815.495,A -85,B 0,C 180,E1 -28809.225,E2 -28809.225} C_VEL
LIN {X 0,Y 100.9,Z 813.806,A -85,B 0,C 180,E1 -28812.807,E2 -28812.807} C_VEL
LIN {X 0,Y 112.668,Z 810.246,A -85,B 0,C 180,E1 -28816.779,E2 -28816.779} C_VEL
LIN {X 0,Y 124.351,Z 805.247,A -85,B 0,C 180,E1 -28819.822,E2 -28819.822} C_VEL
LIN {X 0,Y 127.691,Z 803.581,A -85,B 0,C 180,E1 -28820.668,E2 -28820.668} C_VEL
LIN {X 0,Y 118.019,Z 808.832,A -85,B 0,C 180,E1 -28822.631,E2 -28822.631} C_VEL
LIN {X 0,Y 105.418,Z 814.27,A -85,B 0,C 180,E1 -28825.843,E2 -28825.843} C_VEL
LIN {X 0,Y 96.34,Z 817.334,A -85,B 0,C 180,E1 -28828.91,E2 -28828.91} C_VEL
LIN {X 0,Y 84.997,Z 820.145,A -85,B 0,C 180,E1 -28834.226,E2 -28834.226} C_VEL
LIN {X 0,Y 74.825,Z 821.616,A -85,B 0,C 180,E1 -28841.289,E2 -28841.289} C_VEL
LIN {X 0,Y 66.345,Z 821.777,A -85,B 0,C 180,E1 -28850.537,E2 -28850.537} C_VEL
LIN {X 0,Y 60.197,Z 820.555,A -85,B 0,C 180,E1 -28862.161,E2 -28862.161} C_VEL
LIN {X 0,Y 57.44,Z 818.007,A -85,B 0,C 180,E1 -28875.836,E2 -28875.836} C_VEL
LIN {X 0,Y 57.256,Z 817.283,A -85,B 0,C 180,E1 -28879.517,E2 -28879.517} C_VEL
LIN {X 0,Y 57.018,Z 820.121,A -85,B 0,C 180,E1 -28890,E2 -28890} C_VEL
LIN {X 0,Y 56.527,Z 821.331,A -85,B 0,C 180,E1 -28897.142,E2 -28897.142} C_VEL
LIN {X 0,Y 57.927,Z 822.571,A -85,B 0,C 180,E1 -28911.344,E2 -28911.344} C_VEL
LIN {X 0,Y 59.917,Z 822.618,A -85,B 0,C 180,E1 -28917.981,E2 -28917.981} C_VEL
LIN {X 0,Y 66.162,Z 821.509,A -85,B 0,C 180,E1 -28929.593,E2 -28929.593} C_VEL
LIN {X 0,Y 74.634,Z 818.871,A -85,B 0,C 180,E1 -28938.878,E2 -28938.878} C_VEL
LIN {X 0,Y 82.132,Z 815.798,A -85,B 0,C 180,E1 -28944.38,E2 -28944.38} C_VEL
LIN {X 0,Y 90.357,Z 811.718,A -85,B 0,C 180,E1 -28948.822,E2 -28948.822} C_VEL
LIN {X 0,Y 100.548,Z 805.491,A -85,B 0,C 180,E1 -28953.02,E2 -28953.02} C_VEL
LIN {X 0,Y 109.734,Z 798.756,A -85,B 0,C 180,E1 -28955.871,E2 -28955.871} C_VEL
LIN {X 0,Y 119.183,Z 790.441,A -85,B 0,C 180,E1 -28958.236,E2 -28958.236} C_VEL
LIN {X 0,Y 127.18,Z 781.903,A -85,B 0,C 180,E1 -28959.951,E2 -28959.951} C_VEL
LIN {X 0,Y 135.403,Z 771.414,A -85,B 0,C 180,E1 -28961.303,E2 -28961.303} C_VEL
LIN {X 0,Y 142.007,Z 761.047,A -85,B 0,C 180,E1 -28962.301,E2 -28962.301} C_VEL
LIN {X 0,Y 147.867,Z 749.518,A -85,B 0,C 180,E1 -28963.082,E2 -28963.082} C_VEL
LIN {X 0,Y 153.033,Z 735.982,A -85,B 0,C 180,E1 -28963.754,E2 -28963.754} C_VEL
LIN {X 0,Y 155.729,Z 726.167,A -85,B 0,C 180,E1 -28964.122,E2 -28964.122} C_VEL
LIN {X 0,Y 154.943,Z 723.167,A -85,B 0,C 180,E1 -28967.558,E2 -28967.558} C_VEL
LIN {X 0,Y 154.432,Z 720.707,A -85,B 0,C 180,E1 -28971.495,E2 -28971.495} C_VEL
LIN {X 0,Y 154.248,Z 720.568,A -85,B 0,C 180,E1 -28973.19,E2 -28973.19} C_VEL
LIN {X 0,Y 154.035,Z 721.241,A -85,B 0,C 180,E1 -28974.626,E2 -28974.626} C_VEL
LIN {X 0,Y 153.345,Z 724.306,A -85,B 0,C 180,E1 -28976.82,E2 -28976.82} C_VEL
LIN {X 0,Y 152.593,Z 728.373,A -85,B 0,C 180,E1 -28979.474,E2 -28979.474} C_VEL
LIN {X 0,Y 152.561,Z 729.161,A -85,B 0,C 180,E1 -28980.447,E2 -28980.447} C_VEL
LIN {X 0,Y 152.657,Z 731.243,A -85,B 0,C 180,E1 -28982.968,E2 -28982.968} C_VEL
LIN {X 0,Y 147.918,Z 743.865,A -85,B 0,C 180,E1 -28983.848,E2 -28983.848} C_VEL
LIN {X 0,Y 141.966,Z 755.816,A -85,B 0,C 180,E1 -28984.956,E2 -28984.956} C_VEL
LIN {X 0,Y 135.7,Z 765.701,A -85,B 0,C 180,E1 -28986.141,E2 -28986.141} C_VEL
LIN {X 0,Y 127.662,Z 775.979,A -85,B 0,C 180,E1 -28987.734,E2 -28987.734} C_VEL
LIN {X 0,Y 119.435,Z 784.61,A -85,B 0,C 180,E1 -28989.584,E2 -28989.584} C_VEL
LIN {X 0,Y 109.648,Z 792.971,A -85,B 0,C 180,E1 -28992.193,E2 -28992.193} C_VEL
LIN {X 0,Y 101.71,Z 798.589,A -85,B 0,C 180,E1 -28994.682,E2 -28994.682} C_VEL
LIN {X 0,Y 92.098,Z 804.19,A -85,B 0,C 180,E1 -28998.342,E2 -28998.342} C_VEL
LIN {X 0,Y 83.598,Z 808.152,A -85,B 0,C 180,E1 -29002.372,E2 -29002.372} C_VEL
LIN {X 0,Y 74.191,Z 811.533,A -85,B 0,C 180,E1 -29008.271,E2 -29008.271} C_VEL
LIN {X 0,Y 67.598,Z 813.199,A -85,B 0,C 180,E1 -29013.724,E2 -29013.724} C_VEL
LIN {X 0,Y 63.032,Z 814.018,A -85,B 0,C 180,E1 -29018.696,E2 -29018.696} C_VEL
LIN {X 0,Y 57.062,Z 814.427,A -85,B 0,C 180,E1 -29027.646,E2 -29027.646} C_VEL
LIN {X 0,Y 52.727,Z 813.907,A -85,B 0,C 180,E1 -29037.781,E2 -29037.781} C_VEL
LIN {X 0,Y 50.75,Z 813.06,A -85,B 0,C 180,E1 -29045.453,E2 -29045.453} C_VEL
LIN {X 0,Y 49.698,Z 811.765,A -85,B 0,C 180,E1 -29053.571,E2 -29053.571} C_VEL
LIN {X 0,Y 49.579,Z 809.842,A -85,B 0,C 180,E1 -29062.877,E2 -29062.877} C_VEL
LIN {X 0,Y 50.957,Z 806.697,A -85,B 0,C 180,E1 -29073.954,E2 -29073.954} C_VEL
LIN {X 0,Y 54.152,Z 802.258,A -85,B 0,C 180,E1 -29085.044,E2 -29085.044} C_VEL
LIN {X 0,Y 55.564,Z 800.506,A -85,B 0,C 180,E1 -29088.433,E2 -29088.433} C_VEL
LIN {X 0,Y 53.664,Z 799.006,A -85,B 0,C 180,E1 -29093.546,E2 -29093.546} C_VEL
LIN {X 0,Y 50.736,Z 797.575,A -85,B 0,C 180,E1 -29100.031,E2 -29100.031} C_VEL
LIN {X 0,Y 50.332,Z 797.085,A -85,B 0,C 180,E1 -29102.031,E2 -29102.031} C_VEL
LIN {X 0,Y 49.234,Z 803.504,A -85,B 0,C 180,E1 -29115.538,E2 -29115.538} C_VEL
LIN {X 0,Y 50.256,Z 807.881,A -85,B 0,C 180,E1 -29127.039,E2 -29127.039} C_VEL
LIN {X 0,Y 53.107,Z 811.398,A -85,B 0,C 180,E1 -29137.871,E2 -29137.871} C_VEL
LIN {X 0,Y 57.61,Z 814.036,A -85,B 0,C 180,E1 -29147.4,E2 -29147.4} C_VEL
LIN {X 0,Y 63.455,Z 815.874,A -85,B 0,C 180,E1 -29155.4,E2 -29155.4} C_VEL
LIN {X 0,Y 70.322,Z 816.961,A -85,B 0,C 180,E1 -29162.013,E2 -29162.013} C_VEL
LIN {X 0,Y 77.95,Z 817.287,A -85,B 0,C 180,E1 -29167.373,E2 -29167.373} C_VEL
LIN {X 0,Y 86.143,Z 816.812,A -85,B 0,C 180,E1 -29171.763,E2 -29171.763} C_VEL
LIN {X 0,Y 98.343,Z 814.856,A -85,B 0,C 180,E1 -29176.61,E2 -29176.61} C_VEL
LIN {X 0,Y 108.938,Z 811.986,A -85,B 0,C 180,E1 -29179.811,E2 -29179.811} C_VEL
LIN {X 0,Y 105.727,Z 813.343,A -85,B 0,C 180,E1 -29181.472,E2 -29181.472} C_VEL
LIN {X 0,Y 93.114,Z 817.281,A -85,B 0,C 180,E1 -29185.082,E2 -29185.082} C_VEL
LIN {X 0,Y 81.206,Z 819.818,A -85,B 0,C 180,E1 -29190.069,E2 -29190.069} C_VEL
LIN {X 0,Y 70.332,Z 821.004,A -85,B 0,C 180,E1 -29196.928,E2 -29196.928} C_VEL
LIN {X 0,Y 61.03,Z 820.877,A -85,B 0,C 180,E1 -29206.297,E2 -29206.297} C_VEL
LIN {X 0,Y 54.05,Z 819.433,A -85,B 0,C 180,E1 -29218.661,E2 -29218.661} C_VEL
LIN {X 0,Y 50.646,Z 816.666,A -85,B 0,C 180,E1 -29233.887,E2 -29233.887} C_VEL
LIN {X 0,Y 50.484,Z 816.051,A -85,B 0,C 180,E1 -29236.717,E2 -29236.717} C_VEL
LIN {X 0,Y 49.92,Z 819.356,A -85,B 0,C 180,E1 -29250,E2 -29250} C_VEL
LIN {X 0,Y 49.467,Z 820.614,A -85,B 0,C 180,E1 -29258.168,E2 -29258.168} C_VEL
LIN {X 0,Y 51.35,Z 821.917,A -85,B 0,C 180,E1 -29274.242,E2 -29274.242} C_VEL
LIN {X 0,Y 53.707,Z 822.006,A -85,B 0,C 180,E1 -29281.562,E2 -29281.562} C_VEL
LIN {X 0,Y 60.823,Z 820.979,A -85,B 0,C 180,E1 -29293.889,E2 -29293.889} C_VEL
LIN {X 0,Y 70.14,Z 818.423,A -85,B 0,C 180,E1 -29303.281,E2 -29303.281} C_VEL
LIN {X 0,Y 78.195,Z 815.414,A -85,B 0,C 180,E1 -29308.63,E2 -29308.63} C_VEL
LIN {X 0,Y 86.879,Z 811.408,A -85,B 0,C 180,E1 -29312.85,E2 -29312.85} C_VEL
LIN {X 0,Y 97.528,Z 805.298,A -85,B 0,C 180,E1 -29316.745,E2 -29316.745} C_VEL
LIN {X 0,Y 107.033,Z 798.656,A -85,B 0,C 180,E1 -29319.334,E2 -29319.334} C_VEL
LIN {X 0,Y 116.743,Z 790.458,A -85,B 0,C 180,E1 -29321.466,E2 -29321.466} C_VEL
LIN {X 0,Y 124.928,Z 782.089,A -85,B 0,C 180,E1 -29323.005,E2 -29323.005} C_VEL
LIN {X 0,Y 133.303,Z 771.769,A -85,B 0,C 180,E1 -29324.187,E2 -29324.187} C_VEL
LIN {X 0,Y 140.867,Z 760.209,A -85,B 0,C 180,E1 -29325.153,E2 -29325.153} C_VEL
LIN {X 0,Y 146.776,Z 748.682,A -85,B 0,C 180,E1 -29325.828,E2 -29325.828} C_VEL
LIN {X 0,Y 151.843,Z 735.6,A -85,B 0,C 180,E1 -29326.398,E2 -29326.398} C_VEL
LIN {X 0,Y 153.217,Z 731.037,A -85,B 0,C 180,E1 -29326.585,E2 -29326.585} C_VEL
LIN {X 0,Y 152.862,Z 729.27,A -85,B 0,C 180,E1 -29329.068,E2 -29329.068} C_VEL
LIN {X 0,Y 152.758,Z 727.678,A -85,B 0,C 180,E1 -29331.401,E2 -29331.401} C_VEL
LIN {X 0,Y 152.597,Z 727.424,A -85,B 0,C 180,E1 -29337.69,E2 -29337.69} C_VEL
LIN {X 0,Y 152.561,Z 729.161,A -85,B 0,C 180,E1 -29340.447,E2 -29340.447} C_VEL
LIN {X 0,Y 152.415,Z 730.202,A -85,B 0,C 180,E1 -29341.091,E2 -29341.091} C_VEL
LIN {X 0,Y 151.772,Z 732.5,A -85,B 0,C 180,E1 -29341.579,E2 -29341.579} C_VEL
LIN {X 0,Y 150.475,Z 736.298,A -85,B 0,C 180,E1 -29341.778,E2 -29341.778} C_VEL
LIN {X 0,Y 145.832,Z 746.784,A -85,B 0,C 180,E1 -29341.377,E2 -29341.377} C_VEL
LIN {X 0,Y 144.812,Z 748.821,A -85,B 0,C 180,E1 -29341.474,E2 -29341.474} C_VEL
LIN {X 0,Y 138.275,Z 760.513,A -85,B 0,C 180,E1 -29342.509,E2 -29342.509} C_VEL
LIN {X 0,Y 130.313,Z 771.646,A -85,B 0,C 180,E1 -29343.876,E2 -29343.876} C_VEL
LIN {X 0,Y 121.778,Z 781.27,A -85,B 0,C 180,E1 -29345.439,E2 -29345.439} C_VEL
LIN {X 0,Y 113.342,Z 789.077,A -85,B 0,C 180,E1 -29347.214,E2 -29347.214} C_VEL
LIN {X 0,Y 103.387,Z 796.599,A -85,B 0,C 180,E1 -29349.717,E2 -29349.717} C_VEL
LIN {X 0,Y 93.642,Z 802.576,A -85,B 0,C 180,E1 -29352.67,E2 -29352.67} C_VEL
LIN {X 0,Y 84.182,Z 807.227,A -85,B 0,C 180,E1 -29356.248,E2 -29356.248} C_VEL
LIN {X 0,Y 75.099,Z 810.705,A -85,B 0,C 180,E1 -29360.641,E2 -29360.641} C_VEL
LIN {X 0,Y 69.334,Z 812.431,A -85,B 0,C 180,E1 -29364.18,E2 -29364.18} C_VEL
LIN {X 0,Y 63.841,Z 813.696,A -85,B 0,C 180,E1 -29368.278,E2 -29368.278} C_VEL
LIN {X 0,Y 58.74,Z 814.552,A -85,B 0,C 180,E1 -29373.124,E2 -29373.124} C_VEL
LIN {X 0,Y 51.336,Z 815.039,A -85,B 0,C 180,E1 -29383.197,E2 -29383.197} C_VEL
LIN {X 0,Y 46.75,Z 814.576,A -85,B 0,C 180,E1 -29393.036,E2 -29393.036} C_VEL
LIN {X 0,Y 44.267,Z 813.784,A -85,B 0,C 180,E1 -29401.557,E2 -29401.557} C_VEL
LIN {X 0,Y 42.8,Z 812.538,A -85,B 0,C 180,E1 -29410.828,E2 -29410.828} C_VEL
LIN {X 0,Y 42.489,Z 810.402,A -85,B 0,C 180,E1 -29422.949,E2 -29422.949} C_VEL
LIN {X 0,Y 44.784,Z 806.242,A -85,B 0,C 180,E1 -29439.028,E2 -29439.028} C_VEL
LIN {X 0,Y 48.051,Z 802.395,A -85,B 0,C 180,E1 -29449.205,E2 -29449.205} C_VEL
LIN {X 0,Y 47.159,Z 801.754,A -85,B 0,C 180,E1 -29451.857,E2 -29451.857} C_VEL
LIN {X 0,Y 42.564,Z 799.206,A -85,B 0,C 180,E1 -29466.191,E2 -29466.191} C_VEL
LIN {X 0,Y 42.431,Z 805.336,A -85,B 0,C 180,E1 -29482.086,E2 -29482.086} C_VEL
LIN {X 0,Y 45.506,Z 810.333,A -85,B 0,C 180,E1 -29497.914,E2 -29497.914} C_VEL
LIN {X 0,Y 52.164,Z 814.311,A -85,B 0,C 180,E1 -29512.257,E2 -29512.257} C_VEL
LIN {X 0,Y 58.298,Z 816.229,A -85,B 0,C 180,E1 -29520,E2 -29520} C_VEL
LIN {X 0,Y 65.227,Z 817.43,A -85,B 0,C 180,E1 -29526.186,E2 -29526.186} C_VEL
LIN {X 0,Y 72.803,Z 817.962,A -85,B 0,C 180,E1 -29531.132,E2 -29531.132} C_VEL
LIN {X 0,Y 80.798,Z 817.863,A -85,B 0,C 180,E1 -29535.126,E2 -29535.126} C_VEL
LIN {X 0,Y 93.004,Z 816.464,A -85,B 0,C 180,E1 -29539.647,E2 -29539.647} C_VEL
LIN {X 0,Y 91.37,Z 816.964,A -85,B 0,C 180,E1 -29540.699,E2 -29540.699} C_VEL
LIN {X 0,Y 77.889,Z 819.403,A -85,B 0,C 180,E1 -29545.539,E2 -29545.539} C_VEL
LIN {X 0,Y 66.311,Z 820.323,A -85,B 0,C 180,E1 -29552.021,E2 -29552.021} C_VEL
LIN {X 0,Y 56.113,Z 819.958,A -85,B 0,C 180,E1 -29561.283,E2 -29561.283} C_VEL
LIN {X 0,Y 48.178,Z 818.268,A -85,B 0,C 180,E1 -29574.304,E2 -29574.304} C_VEL
LIN {X 0,Y 43.967,Z 815.209,A -85,B 0,C 180,E1 -29591.356,E2 -29591.356} C_VEL
LIN {X 0,Y 43.805,Z 814.853,A -85,B 0,C 180,E1 -29593.275,E2 -29593.275} C_VEL
LIN {X 0,Y 42.824,Z 818.578,A -85,B 0,C 180,E1 -29610,E2 -29610} C_VEL
LIN {X 0,Y 42.446,Z 819.899,A -85,B 0,C 180,E1 -29619.53,E2 -29619.53} C_VEL
LIN {X 0,Y 44.933,Z 821.26,A -85,B 0,C 180,E1 -29637.983,E2 -29637.983} C_VEL
LIN {X 0,Y 51.503,Z 821.128,A -85,B 0,C 180,E1 -29653.021,E2 -29653.021} C_VEL
LIN {X 0,Y 60.815,Z 819.401,A -85,B 0,C 180,E1 -29663.991,E2 -29663.991} C_VEL
LIN {X 0,Y 66.126,Z 817.965,A -85,B 0,C 180,E1 -29668.237,E2 -29668.237} C_VEL
LIN {X 0,Y 74.738,Z 815.025,A -85,B 0,C 180,E1 -29673.292,E2 -29673.292} C_VEL
LIN {X 0,Y 83.867,Z 811.093,A -85,B 0,C 180,E1 -29677.186,E2 -29677.186} C_VEL
LIN {X 0,Y 93.341,Z 806.054,A -85,B 0,C 180,E1 -29680.245,E2 -29680.245} C_VEL
LIN {X 0,Y 103.09,Z 799.766,A -85,B 0,C 180,E1 -29682.631,E2 -29682.631} C_VEL
LIN {X 0,Y 113.016,Z 791.936,A -85,B 0,C 180,E1 -29684.548,E2 -29684.548} C_VEL
LIN {X 0,Y 121.378,Z 783.985,A -85,B 0,C 180,E1 -29685.89,E2 -29685.89} C_VEL
LIN {X 0,Y 129.842,Z 774.314,A -85,B 0,C 180,E1 -29686.974,E2 -29686.974} C_VEL
LIN {X 0,Y 137.51,Z 763.563,A -85,B 0,C 180,E1 -29687.804,E2 -29687.804} C_VEL
LIN {X 0,Y 144.252,Z 751.574,A -85,B 0,C 180,E1 -29688.442,E2 -29688.442} C_VEL
LIN {X 0,Y 149.33,Z 739.921,A -85,B 0,C 180,E1 -29688.901,E2 -29688.901} C_VEL
LIN {X 0,Y 150.346,Z 737.081,A -85,B 0,C 180,E1 -29689.001,E2 -29689.001} C_VEL
LIN {X 0,Y 150.642,Z 736.032,A -85,B 0,C 180,E1 -29689.245,E2 -29689.245} C_VEL
LIN {X 0,Y 150.603,Z 734.322,A -85,B 0,C 180,E1 -29691.952,E2 -29691.952} C_VEL
LIN {X 0,Y 150.419,Z 734.128,A -85,B 0,C 180,E1 -29697.322,E2 -29697.322} C_VEL
LIN {X 0,Y 150.242,Z 735.977,A -85,B 0,C 180,E1 -29700.39,E2 -29700.39} C_VEL
LIN {X 0,Y 149.698,Z 737.548,A -85,B 0,C 180,E1 -29700.693,E2 -29700.693} C_VEL
LIN {X 0,Y 144.812,Z 748.821,A -85,B 0,C 180,E1 -29701.474,E2 -29701.474} C_VEL
LIN {X 0,Y 142.943,Z 752.384,A -85,B 0,C 180,E1 -29701.503,E2 -29701.503} C_VEL
LIN {X 0,Y 139.539,Z 757.967,A -85,B 0,C 180,E1 -29700.821,E2 -29700.821} C_VEL
LIN {X 0,Y 135.887,Z 763.412,A -85,B 0,C 180,E1 -29700.123,E2 -29700.123} C_VEL
LIN {X 0,Y 133.595,Z 766.644,A -85,B 0,C 180,E1 -29700.159,E2 -29700.159} C_VEL
LIN {X 0,Y 124.784,Z 777.452,A -85,B 0,C 180,E1 -29701.451,E2 -29701.451} C_VEL
LIN {X 0,Y 116.107,Z 786.086,A -85,B 0,C 180,E1 -29702.896,E2 -29702.896} C_VEL
LIN {X 0,Y 105.808,Z 794.353,A -85,B 0,C 180,E1 -29704.928,E2 -29704.928} C_VEL
LIN {X 0,Y 95.66,Z 800.939,A -85,B 0,C 180,E1 -29707.342,E2 -29707.342} C_VEL
LIN {X 0,Y 85.709,Z 806.116,A -85,B 0,C 180,E1 -29710.279,E2 -29710.279} C_VEL
LIN {X 0,Y 76.006,Z 810.053,A -85,B 0,C 180,E1 -29713.864,E2 -29713.864} C_VEL
LIN {X 0,Y 66.685,Z 812.886,A -85,B 0,C 180,E1 -29718.468,E2 -29718.468} C_VEL
LIN {X 0,Y 60.736,Z 814.192,A -85,B 0,C 180,E1 -29722.228,E2 -29722.228} C_VEL
LIN {X 0,Y 49.865,Z 815.575,A -85,B 0,C 180,E1 -29732.262,E2 -29732.262} C_VEL
LIN {X 0,Y 45.209,Z 815.611,A -85,B 0,C 180,E1 -29738.989,E2 -29738.989} C_VEL
LIN {X 0,Y 38.046,Z 814.489,A -85,B 0,C 180,E1 -29756.347,E2 -29756.347} C_VEL
LIN {X 0,Y 36.062,Z 813.308,A -85,B 0,C 180,E1 -29767.06,E2 -29767.06} C_VEL
LIN {X 0,Y 35.397,Z 810.952,A -85,B 0,C 180,E1 -29783.098,E2 -29783.098} C_VEL
LIN {X 0,Y 37.735,Z 807.154,A -85,B 0,C 180,E1 -29800.734,E2 -29800.734} C_VEL
LIN {X 0,Y 39.049,Z 805.716,A -85,B 0,C 180,E1 -29805.662,E2 -29805.662} C_VEL
LIN {X 0,Y 40.229,Z 804.201,A -85,B 0,C 180,E1 -29810.45,E2 -29810.45} C_VEL
LIN {X 0,Y 35.099,Z 801.349,A -85,B 0,C 180,E1 -29831.337,E2 -29831.337} C_VEL
LIN {X 0,Y 35.093,Z 801.322,A -85,B 0,C 180,E1 -29832.423,E2 -29832.423} C_VEL
LIN {X 0,Y 36.397,Z 807.063,A -85,B 0,C 180,E1 -29851.143,E2 -29851.143} C_VEL
LIN {X 0,Y 40.068,Z 810.904,A -85,B 0,C 180,E1 -29864.746,E2 -29864.746} C_VEL
LIN {X 0,Y 48.59,Z 815.058,A -85,B 0,C 180,E1 -29880,E2 -29880} C_VEL
LIN {X 0,Y 56.809,Z 817.175,A -85,B 0,C 180,E1 -29888.242,E2 -29888.242} C_VEL
LIN {X 0,Y 65.156,Z 818.343,A -85,B 0,C 180,E1 -29893.891,E2 -29893.891} C_VEL
LIN {X 0,Y 76.011,Z 818.713,A -85,B 0,C 180,E1 -29899.047,E2 -29899.047} C_VEL
LIN {X 0,Y 75.094,Z 818.973,A -85,B 0,C 180,E1 -29900.631,E2 -29900.631} C_VEL
LIN {X 0,Y 62.578,Z 819.599,A -85,B 0,C 180,E1 -29906.694,E2 -29906.694} C_VEL
LIN {X 0,Y 51.708,Z 818.949,A -85,B 0,C 180,E1 -29915.364,E2 -29915.364} C_VEL
LIN {X 0,Y 42.658,Z 816.994,A -85,B 0,C 180,E1 -29928.778,E2 -29928.778} C_VEL
LIN {X 0,Y 37.299,Z 813.658,A -85,B 0,C 180,E1 -29948.661,E2 -29948.661} C_VEL
LIN {X 0,Y 36.021,Z 815.872,A -85,B 0,C 180,E1 -29958.749,E2 -29958.749} C_VEL
LIN {X 0,Y 35.73,Z 817.796,A -85,B 0,C 180,E1 -29970,E2 -29970} C_VEL
LIN {X 0,Y 35.448,Z 819.159,A -85,B 0,C 180,E1 -29981.435,E2 -29981.435} C_VEL
LIN {X 0,Y 38.78,Z 820.604,A -85,B 0,C 180,E1 -30002.933,E2 -30002.933} C_VEL
LIN {X 0,Y 46.54,Z 820.546,A -85,B 0,C 180,E1 -30019.027,E2 -30019.027} C_VEL
LIN {X 0,Y 51.481,Z 819.926,A -85,B 0,C 180,E1 -30024.993,E2 -30024.993} C_VEL
LIN {X 0,Y 62.67,Z 817.507,A -85,B 0,C 180,E1 -30033.781,E2 -30033.781} C_VEL
LIN {X 0,Y 71.816,Z 814.636,A -85,B 0,C 180,E1 -30038.382,E2 -30038.382} C_VEL
LIN {X 0,Y 81.373,Z 810.778,A -85,B 0,C 180,E1 -30041.809,E2 -30041.809} C_VEL
LIN {X 0,Y 91.185,Z 805.819,A -85,B 0,C 180,E1 -30044.451,E2 -30044.451} C_VEL
LIN {X 0,Y 101.197,Z 799.62,A -85,B 0,C 180,E1 -30046.473,E2 -30046.473} C_VEL
LIN {X 0,Y 111.34,Z 791.939,A -85,B 0,C 180,E1 -30048.06,E2 -30048.06} C_VEL
LIN {X 0,Y 121.545,Z 782.348,A -85,B 0,C 180,E1 -30049.404,E2 -30049.404} C_VEL
LIN {X 0,Y 130.161,Z 772.466,A -85,B 0,C 180,E1 -30050.191,E2 -30050.191} C_VEL
LIN {X 0,Y 137.924,Z 761.326,A -85,B 0,C 180,E1 -30050.838,E2 -30050.838} C_VEL
LIN {X 0,Y 144.438,Z 749.56,A -85,B 0,C 180,E1 -30051.316,E2 -30051.316} C_VEL
LIN {X 0,Y 147.611,Z 742.455,A -85,B 0,C 180,E1 -30051.548,E2 -30051.548} C_VEL
LIN {X 0,Y 148.051,Z 741.235,A -85,B 0,C 180,E1 -30051.813,E2 -30051.813} C_VEL
LIN {X 0,Y 147.861,Z 740.761,A -85,B 0,C 180,E1 -30056.495,E2 -30056.495} C_VEL
LIN {X 0,Y 147.839,Z 740.915,A -85,B 0,C 180,E1 -30057.275,E2 -30057.275} C_VEL
LIN {X 0,Y 147.66,Z 741.554,A -85,B 0,C 180,E1 -30058.16,E2 -30058.16} C_VEL
LIN {X 0,Y 142.329,Z 752.744,A -85,B 0,C 180,E1 -30058.915,E2 -30058.915} C_VEL
LIN {X 0,Y 135.857,Z 763.389,A -85,B 0,C 180,E1 -30059.808,E2 -30059.808} C_VEL
LIN {X 0,Y 133.595,Z 766.644,A -85,B 0,C 180,E1 -30060.159,E2 -30060.159} C_VEL
LIN {X 0,Y 130.029,Z 771.334,A -85,B 0,C 180,E1 -30060.388,E2 -30060.388} C_VEL
LIN {X 0,Y 123.473,Z 778.741,A -85,B 0,C 180,E1 -30059.998,E2 -30059.998} C_VEL
LIN {X 0,Y 116.38,Z 785.63,A -85,B 0,C 180,E1 -30059.605,E2 -30059.605} C_VEL
LIN {X 0,Y 111.959,Z 789.431,A -85,B 0,C 180,E1 -30059.917,E2 -30059.917} C_VEL
LIN {X 0,Y 101.944,Z 796.858,A -85,B 0,C 180,E1 -30061.626,E2 -30061.626} C_VEL
LIN {X 0,Y 91.557,Z 803.021,A -85,B 0,C 180,E1 -30063.743,E2 -30063.743} C_VEL
LIN {X 0,Y 81.32,Z 807.843,A -85,B 0,C 180,E1 -30066.355,E2 -30066.355} C_VEL
LIN {X 0,Y 71.277,Z 811.48,A -85,B 0,C 180,E1 -30069.605,E2 -30069.605} C_VEL
LIN {X 0,Y 64.04,Z 813.498,A -85,B 0,C 180,E1 -30072.679,E2 -30072.679} C_VEL
LIN {X 0,Y 52.225,Z 815.616,A -85,B 0,C 180,E1 -30079.613,E2 -30079.613} C_VEL
LIN {X 0,Y 46.388,Z 816.143,A -85,B 0,C 180,E1 -30084.632,E2 -30084.632} C_VEL
LIN {X 0,Y 41,Z 816.251,A -85,B 0,C 180,E1 -30091.012,E2 -30091.012} C_VEL
